Omron CX-Programmer project COREX_92 (CX-Programmer 9.20)
; (V2.0)

# PLC NewPLC1: CJ1G-H CPU42
I/O table (CPU CJ1G-CPU42H): rack 0 slot 0 CJ1W-ID261; rack 0 slot 1 CJ1W-ID261; rack 0 slot 2 CJ1W-OD211; rack 0 slot 3 CJ1W-OD212; rack 0 slot 4 CJ1W-OD212; rack 0 slot 5 CJ1W-OD212; rack 0 slot 6 CJ1W-OD212; rack 0 slot 7 CJ1W-OD212; rack 0 slot 8 CJ1W-AD041-V1

## Global symbols (name address type ; comment)
2000 CHANNEL  ; Peak Value Hold Unitat 0
2001 CHANNEL  ; AIn1 - cèlula aliniador MUW
2002 CHANNEL  ; AIn2 - cèlula ultrassons reb. esquerra
2003 CHANNEL  ; AIn3 - cèlula aliniador reb. dret
2009 CHANNEL  ; Detecció Desconnexió Entrades Unitat 0
2.05 BOOL  ; Relé velocitat màquina mestre
2.06 BOOL  ; màquina mestra unida
2.07 BOOL  ; Info reset de la mestra cap a l'esclava
2.08 BOOL  ; Marxa des de la mestra
2.09 BOOL  ; Mestra en marxa en mode B (Engegada de la mestra)
2.10 BOOL  ; premarxa de la mestra
2.11 BOOL  ; $?St$Bk?_#[971] / mestre en mode "A"$?St$Bk?_#[971]
2.12 BOOL  ; Sèrie de paros de la mestra
2.13 BOOL  ; Màquina mestra en cicle
2.14 BOOL  ; Info SM alt a master
2.15 BOOL  ; Relé velocitat mestra a esclava
30.06 BOOL  ; Sel. Giro Invers MUW
30.07 BOOL  ; Puls.Tensat MUW
320.09 BOOL  ; Tecla calibrar ultrassons MUW
320.10 BOOL  ; Tecla calibrar ultrassons reb.esquerra
320.11 BOOL  ; Tecla calibrar ultrassons reb. dret
32.03 BOOL  ; Alarma variadors de freqüència
32.07 BOOL  ; Marxa aliniador desbobinador
34.13 BOOL  ; Botó negre comanament a distància
36.01 BOOL  ; Selector mode desplaçador (abans selector línia)
36.03 BOOL  ; Detector SM alt master
36.04 BOOL  ; Detector SM de la mestra al mig
36.05 BOOL  ; Detector SM baix master
36.06 BOOL  ; Pulsador marxa lenta SM
36.08 BOOL  ; Detector SM alt esclava
36.09 BOOL  ; Detector SM baix esclava
36.10 BOOL  ; Màquina esclava unida
36.11 BOOL  ; Pulsador de reset de la esclava
36.12 BOOL  ; Condicions premarxa esclava
36.13 BOOL  ; Esclava en premarxa
36.14 BOOL  ; $?St$Bk?_#[972] / esclava en mode "A"$?St$Bk?_#[972]
36.15 BOOL  ; Sèrie de paros de l'esclava
37.00 BOOL  ; Màquina esclava en cicle
4.12 BOOL  ; elv desplaçar a l'esquerra aliniador desbobinador
4.13 BOOL  ; elv desplaçar a la dreta aliniador desbobinador
50.05 BOOL  ; Reset des de l'esclava
50.06 BOOL  ; Impuls reset des de l'esclava
5.06 BOOL  ; Pilot MUW
6.14 BOOL  ; Marxa Inversa MUW
7.08 BOOL  ; elv.desplaçar a l'esquerra aliniador esquerra (destapar)
7.09 BOOL  ; elv.desplaçar a la dreta aliniador esquerra (tapar)
7.10 BOOL  ; elv.desplaçar a l'esquerra aliniador dret (tapar)
7.11 BOOL  ; elv.desplaçar a la dreta aliniador dret (destapar)
7.12 BOOL  ; Marxa normal SM
7.13 BOOL  ; Marxa lenta SM
7.14 BOOL  ; contactor motor bufador SM
80.01 BOOL  ; Estat 1 reb. esquerra
80.02 BOOL  ; Estat2 reb. esquerra
80.03 BOOL  ; Estat3 reb. esquerra
81.01 BOOL  ; Estat 1 reb. dret
81.02 BOOL  ; Estat2 reb. dret
81.03 BOOL  ; Estat3 reb. dret
89.00 BOOL  ; aux. detectors SM alt
89.01 BOOL  ; Aux SM baix
89.02 BOOL  ; Aux SM alt
91.10 BOOL  ; Impuls canvi rotlle rebuig
91.11 BOOL  ; Màquines unides
91.12 BOOL  ; Coincidència selecció entre les dues màquines
91.13 BOOL  ; Missatge cal rearmar la màquina esclava
91.14 BOOL  ; Aux.esclava no està en condicions de marxa
91.15 BOOL  ; Aux.Autogir
92.03 BOOL  ; Aux. MUW OK
9.04 BOOL  ; ZIG-ZAG ESQUERRA
9.05 BOOL  ; ZIG-ZAG DRETA
C0032 BOOL  ; nombre bosses rebuig en engegar
C0150 BOOL  ; pulsos aliniador muw
C0151 BOOL  ; Afegit per a variar el punt esquerra
C0152 BOOL  ; Afegit per a variar el punt dret
C0250 BOOL  ; Bosses fabricades x 1E0
C0251 BOOL  ; Bosses fabricades x 1E4
C0252 BOOL  ; Bosses fabricades x 1E8
C0253 BOOL  ; Rotlles esquerres x 1E0
C0254 BOOL  ; Rotlles esquerres x 1E4
C0255 BOOL  ; Rotlles esquerres x 1E8
C0256 BOOL  ; Rotlles drets x 1E0
C0257 BOOL  ; Rotlles drets x 1E4
C0258 BOOL  ; Rotlles drets x 1E8
C0555 BOOL  ; ret
C151 CHANNEL  ; Afegit per a variar ventall cada cicle
D200 CHANNEL  ; Divisor per a l'entrada ultrassonic MUW
D20000 CHANNEL  ; Habilitar conversions Unitat 0
D20001 CHANNEL  ; Configuracio rangs Unitat 0
D20002 CHANNEL  ; Valor mig entrada 1
D20003 CHANNEL  ; Valor mig entrada 2
D20004 CHANNEL  ; Valor mig entrada 3
D20005 CHANNEL  ; Valor mig entrada 4
D20006 CHANNEL  ; Valor mig entrada 5
D20007 CHANNEL  ; Valor mig entrada 6
D20008 CHANNEL  ; Valor mig entrada 7
D20009 CHANNEL  ; Valor mig entrada 8
D20018 CHANNEL  ; Temps conversió/ressolució unitat0
D201 CHANNEL  ; residu divisió
D202 CHANNEL  ; Divisor per a ultrassonic reb. esquerra
D203 CHANNEL  ; residu divisió
D204 CHANNEL  ; Divisor per a ultrassonic reb. dret
D205 CHANNEL  ; residu divisió
D210 CHANNEL  ; Percentatge de lectura del MUW
D220 CHANNEL  ; Percentatge de lectura del reb. esquerra
D222 CHANNEL  ; Quantitat de ventall esquerra (BCD)
D223 CHANNEL  ; Ventall total a fer reb. esquerra
D230 CHANNEL  ; Percentatge de lectura del reb. dret
D232 CHANNEL  ; Quantitat de ventall dret(BCD)
D233 CHANNEL  ; Ventall total a fer reb. dret
D40 CHANNEL  ; missatge a veure en prova pneumàtica
H0.15 BOOL  ; habilita canvi rotlle de rebuig
T0030 BOOL  ; Fi marxa vibrador esquerra
T0031 BOOL  ; Fi marxa vibrador dreta
T0081 BOOL  ; Retard missatge esclava no preparada
T0150 BOOL  ; retard calibrar ultrasons MUW
T0151 BOOL  ; retard calibrar ultrassons reb.esquerra
T0152 BOOL  ; retard calibrar ultrassons reb. dret
T0153 BOOL  ; retard seguretat moviment brusc aliniador MUW
T0154 BOOL  ; temps mínim elv a esquerres desactivada
T0155 BOOL  ; temps mínim elv a dretes desactivada
T0156 BOOL  ; Temps ventall reb. esquerra
T0157 BOOL  ; Temps Interior esquerra (esperem per destapar)
T0158 BOOL  ; Temps ventall reb. dret
T0159 BOOL  ; Temps Interior dret (esperem per destapar)
T0340 BOOL  ; Temps coincidència entre màquines
T0341 BOOL  ; Bufat allargat SM
T0555 BOOL  ; ret
n120_08 120.08 BOOL  ; MSG.DIGIT.0
n120_09 120.09 BOOL  ; MSG.DIGIT.1
n120_10 120.10 BOOL  ; MSG.DIGIT.2
n120_11 120.11 BOOL  ; MSG.DIGIT.3
n120_12 120.12 BOOL  ; MSG.DIGIT.4
n120_13 120.13 BOOL  ; MSG.DIGIT.5
n120_14 120.14 BOOL  ; MSG.DIGIT.6
n235_05 235.05 BOOL  ; CELUL.ROLL.EN VI
n235_06 235.06 BOOL  ; CELUL.VOLC.VAC.I
n236_05 236.05 BOOL  ; CULUL,ROLL.EN.VD
n236_06 236.06 BOOL  ; CELUL.VOLC.VAC.D
n237_00 237.00 BOOL  ; CELUL.DEP/MDR.I
n237_01 237.01 BOOL  ; CELUL.ASCN.LLN.I
n237_05 237.05 BOOL  ; CELUL.R.CAIDO IZ
n237_08 237.08 BOOL  ; CELUL.DEP/MDR.D
n237_09 237.09 BOOL  ; CELUL.ASCN.LLN.D
n237_13 237.13 BOOL  ; CELUL.R.CAIDO DR
n253_08 A402.04 BOOL  ; LOW BATTERY
n253_13 CF113 BOOL  ; ON.
n253_14 CF114 BOOL  ; OFF.
n253_15 A200.15 BOOL  ; FIRST CYCLE FLAG
n254_00 CF104 BOOL  ; IMP 1Min.
n255_00 CF100 BOOL  ; IMP 0.1Seg.
n255_01 CF101 BOOL  ; IMP 0.2Seg
n255_02 CF102 BOOL  ; IMP 1Seg.
n2_00 2.00 BOOL  ; CONTROL VELO.A.I
n2_01 2.01 BOOL  ; CONTROL VELO.B.I
n2_02 2.02 BOOL  ; CONTROL VELO.A.D
n2_03 2.03 BOOL  ; CONTROL VELO.B.D
n2_04 2.04 BOOL  ; RESET INTEGRADOR
n300_00 300.00 BOOL  ; CAMBIO CICLO
n301_00 301.00 BOOL  ; MARCHA/PARO
n301_01 301.01 BOOL  ; CLOCK
n301_02 301.02 BOOL  ; PULSO FLIP-FLOP
n301_03 301.03 BOOL  ; FLIP-FLOP
n301_04 301.04 BOOL  ; RESET
n301_05 301.05 BOOL  ; SET
n302_00 302.00 BOOL  ; SHFT-PISON
n302_01 302.01 BOOL  ; SHFT-EXTRACTOR
n302_02 302.02 BOOL  ; SHFT-VOLCADOR
n302_03 302.03 BOOL  ; SHFT-ASCENSOR
n302_04 302.04 BOOL  ; SHFT-INTRODUCTOR
n302_05 302.05 BOOL  ; SHFT-SOPLADOR
n302_06 302.06 BOOL  ; SHFT-RESET
n303_11 303.11 BOOL  ; I.CIERRE PISONES
n303_12 303.12 BOOL  ; AUX.C.SOPLADORES
n303_13 303.13 BOOL  ; AUX.C.SOPLADORS
n303_14 303.14 BOOL  ; AUX.A.SOPLADORS
n304_00 304.00 BOOL  ; KEEP PI.NEUMATIC
n305_00 305.00 BOOL  ; KEEP 2PI
n305_01 305.01 BOOL  ; I.REPET.2PI
n307_00 307.00 BOOL  ; I.ABRIR PSN.I.
n307_01 307.01 BOOL  ; I.ABRIR PSN.D.
n307_02 307.02 BOOL  ; I.2PI.ABRIR PSN.
n307_03 307.03 BOOL  ; I.1PI.ABRIR PSN.
n307_04 307.04 BOOL  ; I.1PI.CERRAR PSN
n307_05 307.05 BOOL  ; I.CERR.EXTR.I.
n307_06 307.06 BOOL  ; I.CERR.EXTR.D.
n307_07 307.07 BOOL  ; I.2PI CERR.EXTRC
n307_08 307.08 BOOL  ; I.1PI CERR.EXTRC
n307_09 307.09 BOOL  ; I.ABRIR.EXTRACT
n307_10 307.10 BOOL  ; I.2PI ABRIR EXTR
n307_11 307.11 BOOL  ; I.1PI ABRIR EXTR
n307_12 307.12 BOOL  ; I.ABRIR INTRO.I
n307_13 307.13 BOOL  ; I.ABRIR INTRO.D
n307_14 307.14 BOOL  ; I.2PI ABRIR INTR
n307_15 307.15 BOOL  ; I.1PI ABRIR INTR
n308_00 308.00 BOOL  ; KEEP ABRIR PSN.
n308_01 308.01 BOOL  ; KEEP CERRAR PSN.
n308_02 308.02 BOOL  ; KEEP CERRAR EXTR
n308_03 308.03 BOOL  ; KEEP ABRIR EXTRT
n308_04 308.04 BOOL  ; KEEP ABRIR INTRO
n308_05 308.05 BOOL  ; KEEP ABRIR SOPLD
n308_06 308.06 BOOL  ; KEEP CERRAR SOPD
n308_07 308.07 BOOL  ; KEEP BUFA PEINAR
n308_08 308.08 BOOL  ; KEEP BUFA CORTAR
n308_09 308.09 BOOL  ; KEEP MARCHA PITO
n308_10 308.10 BOOL  ; KEEP PRESOSTATO
n309_00 309.00 BOOL  ; I.ABRIR.SOPLADO
n309_01 309.01 BOOL  ; I.2PI.SOPLADO
n309_02 309.02 BOOL  ; I.1PI.SOPLADO
n309_03 309.03 BOOL  ; I.CERR.SOPLADO
n309_04 309.04 BOOL  ; I.2PI.CERR.SOPLD
n309_05 309.05 BOOL  ; I.1PI.CERR.SOPLD
n309_06 309.06 BOOL  ; I.KEEP B.PEINE
n309_07 309.07 BOOL  ; I.KEEP B.CORTE
n309_08 309.08 BOOL  ; _
n309_09 309.09 BOOL  ; I.ELV.GENERAL
n309_10 309.10 BOOL  ; I.2PI.ELV.GENERL
n309_11 309.11 BOOL  ; I.1PI.ELV.GENERL
n309_12 309.12 BOOL  ; I.PRESOSTATO
n309_13 309.13 BOOL  ; KEEP PITO PRESST
n30_00 30.00 BOOL  ; PARO FIN BOBINA
n30_01 30.01 BOOL  ; AVISO FIN BOBINA
n30_02 30.02 BOOL  ; PARO MAT.CORTADO
n30_03 30.03 BOOL  ; COMP.MUW.ALTO
n30_04 30.04 BOOL  ; COMP.MUW.BAJO
n30_05 30.05 BOOL  ; Sel. Giro Normal MUW
n30_08 30.08 BOOL  ; DETECT.GIRO SR
n30_09 30.09 BOOL  ; MARCHA CALOR SR.
n30_10 30.10 BOOL  ; $?St$Bk?_#[973] / SELECTOR "0" SR.$?St$Bk?_#[973]
n30_11 30.11 BOOL  ; $?St$Bk?_#[974] / SELECTOR "MAN"SR$?St$Bk?_#[974]
n30_12 30.12 BOOL  ; ALARM.TEMPE.SR.
n30_13 30.13 BOOL  ; DETECT.COMP.1
n30_14 30.14 BOOL  ; DETECT.COMP.2
n30_15 30.15 BOOL  ; DETEC.CONTADOR
n310_00 310.00 BOOL  ; PULSO CAMBIO PRG
n310_01 310.01 BOOL  ; KEEP CAMBIO PRG
n311_00 311.00 BOOL  ; I.V.CEL.3505
n311_01 311.01 BOOL  ; I.V.CEL.3506
n311_02 311.02 BOOL  ; I.V.CEL.3605
n311_03 311.03 BOOL  ; I.V.CEL.3606
n311_04 311.04 BOOL  ; I.V.CEL.3700
n311_05 311.05 BOOL  ; I.V.CEL.3701
n311_06 311.06 BOOL  ; I.V.CEL.3705
n311_07 311.07 BOOL  ; I.V.CEL.3708
n311_08 311.08 BOOL  ; I.V.CEL.3709
n311_09 311.09 BOOL  ; I.V.CEL.3713
n311_14 311.14 BOOL  ; KEEP PIT.CEL
n311_15 311.15 BOOL  ; I.PITO.V.CEL
n31_00 31.00 BOOL  ; DET.ALTR.COMP3.I, alrma si no el veu
n31_01 31.01 BOOL  ; DETEC.COMP.I. MEDIO para motors
n31_02 31.02 BOOL  ; PULSAD.GIR.PNZ.I
n31_03 31.03 BOOL  ; DET.ALTR.COMP3.D, alarma si no el veu
n31_04 31.04 BOOL  ; DETEC.COMP.D. MEDIO para motors
n31_05 31.05 BOOL  ; DET.VELO.LINEAL
n31_06 31.06 BOOL  ; PULSAD.GIR.PNZ.D
n31_07 31.07 BOOL  ; PRESOST.CADENAS
n31_08 31.08 BOOL  ; $?St$Bk?_#[975] / SELECT.1-2-4 "1"$?St$Bk?_#[975]
n31_09 31.09 BOOL  ; $?St$Bk?_#[976] / SELECT.1-2-4 "4"$?St$Bk?_#[976]
n31_10 31.10 BOOL  ; SEL.CELUL.REGIST
n31_11 31.11 BOOL  ; PULS.AVANC.REGTR
n31_12 31.12 BOOL  ; PULS.RETRO.REGTR
n31_13 31.13 BOOL  ; SE¥AL REGISTR.OK
n31_14 31.14 BOOL  ; SE¥AL ELV RETROC
n31_15 31.15 BOOL  ; SE¥AL ELV.AVANCE
n320_00 320.00 BOOL  ; TECLA + PRESEL
n320_01 320.01 BOOL  ; TECLA - PRESEL
n320_02 320.02 BOOL  ; TECLA RST PRESEL
n320_03 320.03 BOOL  ; TECLA RST.TOT.R.
n320_04 320.04 BOOL  ; TECLA + PRECAL.
n320_05 320.05 BOOL  ; TECLA - PRECAL.
n320_06 320.06 BOOL  ; TECLA PISTA I
n320_07 320.07 BOOL  ; TECLA PISTA I+D
n320_08 320.08 BOOL  ; TECLA PISTA D
n32_00 32.00 BOOL  ; Emergència Principal OK
n32_01 32.01 BOOL  ; SENYAL RELEs STOPs (Preventa Tapa Tambor)
n32_02 32.02 BOOL  ; Magnetotèrmics i disjuntors
n32_04 32.04 BOOL  ; PRESOSTATO
n32_05 32.05 BOOL  ; AJUST.NIV.COMP3I
n32_06 32.06 BOOL  ; AJUST.NIV.COMP3D
n32_08 32.08 BOOL  ; $?St$Bk?_#[977] / SELECT.MODO"A-B"$?St$Bk?_#[977]
n32_09 32.09 BOOL  ; PULSD.RESTART
n32_10 32.10 BOOL  ; PULSD.RESET
n32_11 32.11 BOOL  ; PULSAD.MARCHA
n32_12 32.12 BOOL  ; PULSAD.PARO
n32_13 32.13 BOOL  ; PULSAD.GIR.TAMB.
n32_14 32.14 BOOL  ; ALARMA RESISTRON
n33_00 33.00 BOOL  ; DETEC.C.PISN.I.C
n33_01 33.01 BOOL  ; DETEC.MAX.ROLL.I
n33_02 33.02 BOOL  ; DETEC.C.EXTR.I.A
n33_03 33.03 BOOL  ; DETEC.C.EXTR.I.C
n33_04 33.04 BOOL  ; CELUL.ROLL.EN VI
n33_05 33.05 BOOL  ; CELUL.VOLC.VAC.I
n33_06 33.06 BOOL  ; DETEC.EJE/MNDR.I
n33_07 33.07 BOOL  ; CELUL.DEP/MDR.I
n33_08 33.08 BOOL  ; CELUL.ASCN.LLN.I
n33_09 33.09 BOOL  ; DETEC.C.INTR.I.A
n33_10 33.10 BOOL  ; CELUL.R.CAIDO IZ
n33_11 33.11 BOOL  ; DETEC.C.PISN.D.C
n33_12 33.12 BOOL  ; DETEC.MAX.ROLL.D
n33_13 33.13 BOOL  ; DETEC.C.EXTR.D.A
n33_14 33.14 BOOL  ; DETEC.C.EXTR.D.C
n33_15 33.15 BOOL  ; CULUL,ROLL.EN.VD
n34_00 34.00 BOOL  ; CELUL.VOLC.VAC.D
n34_01 34.01 BOOL  ; DETEC.EJE/MNDR.D
n34_02 34.02 BOOL  ; DETEC.C.SOPLAD.A
n34_03 34.03 BOOL  ; DETEC.C.SOPLAD.C
n34_04 34.04 BOOL  ; CELUL.DEP/MDR.D
n34_05 34.05 BOOL  ; CELUL.ASCN.LLN.D
n34_06 34.06 BOOL  ; DETEC.C.INTR.D.A
n34_07 34.07 BOOL  ; CELUL.R.CAIDO DR
n34_08 34.08 BOOL  ; DETEC.PARO TAMB.
n34_09 34.09 BOOL  ; DETEC.CUADR.TAMB
n34_10 34.10 BOOL  ; DETEC.POSIC.TAMB
n35_00 35.00 BOOL  ; SELEC.MARCHA F.B
n35_01 35.01 BOOL  ; DETECT.F.B.ALTO
n35_02 35.02 BOOL  ; DETECT.F.B.BAJO
n35_03 35.03 BOOL  ; P.MARCH.LENTA FB
n3_00 3.00 BOOL  ; ELV.S.R.
n3_01 3.01 BOOL  ; ELV.SOPLAD.TAMBR
n3_02 3.02 BOOL  ; ELV.ASCENSOR A.I
n3_03 3.03 BOOL  ; ELV.ASCENSOR C.I
n3_04 3.04 BOOL  ; ELV.INTRODUC.A.I
n3_05 3.05 BOOL  ; ELV.INTRODUC.C.I
n3_06 3.06 BOOL  ; ELV. PISON A.I.
n3_07 3.07 BOOL  ; ELV.PISON C.I.
n3_08 3.08 BOOL  ; ELV.EXTRACT.A.I.
n3_09 3.09 BOOL  ; ELV.EXTRACT.C.I.
n3_10 3.10 BOOL  ; ELV.VOLCD.A.I.
n3_11 3.11 BOOL  ; ELV.VOLCD.C.I.
n3_12 3.12 BOOL  ; ELV.SOPLADOR I.
n3_13 3.13 BOOL  ; ELV.BAR SOPLAD.A
n3_14 3.14 BOOL  ; ELV.BAR.SOPLAD.C
n3_15 3.15 BOOL  ; ELV.ACERCADORES
n41_00 41.00 BOOL  ; PRE.POSC-GIR.TAM
n41_01 41.01 BOOL  ; AUX.G.MAN.TAMBOR
n41_02 41.02 BOOL  ; I.POSIC.CILINDRS
n41_03 41.03 BOOL  ; GIRO AUTO TAMBOR
n41_04 41.04 BOOL  ; DETEC.POSICIONAD
n41_05 41.05 BOOL  ; PRE-POSICIONADO
n41_06 41.06 BOOL  ; CLAXON GIRO.TAMB
n41_07 41.07 BOOL  ; PRE-POS.CILINDRO
n41_08 41.08 BOOL  ; CLAXON PREPOS.CL
n42_00 42.00 BOOL  ; CONDIC. EN 0
n42_01 42.01 BOOL  ; CONDIC.EN 2
n42_02 42.02 BOOL  ; I.POSICION TAMB.
n42_03 42.03 BOOL  ; I.EXTRC.PREMARCH
n42_04 42.04 BOOL  ; I.FI.G/TAMBOR
n42_05 42.05 BOOL  ; I.PIS+SOPL.CERRD
n42_06 42.06 BOOL  ; CONDIC.EN 9
n42_07 42.07 BOOL  ; CONDIC.EN 10
n42_08 42.08 BOOL  ; MF.CAX.GIR.TAMB
n42_09 42.09 BOOL  ; MF.CAX.VIBRD.IZD
n42_10 42.10 BOOL  ; MF.CAX.VIBRAD.DR
n42_11 42.11 BOOL  ; CLAX.DEPOSITOS V
n42_15 42.15 BOOL  ; AUX PULD.GIR.TAM
n43_00 43.00 BOOL  ; I.DETEC.C.EXTR.I
n43_01 43.01 BOOL  ; AUX.RET.EXT.I.
n43_02 43.02 BOOL  ; I.RET.EXTRAC.I.
n43_03 43.03 BOOL  ; I.DET.C.EXTRC.D.
n43_04 43.04 BOOL  ; AUX.RET.EXTRAC.D
n43_05 43.05 BOOL  ; I.RET.EXTRAC.D.
n43_06 43.06 BOOL  ; MEMO.MANDRIL IZ.
n43_07 43.07 BOOL  ; I.INTROD.MANDR.I
n43_08 43.08 BOOL  ; MEMO.MANDRIL D.
n43_09 43.09 BOOL  ; I.INTRD.MANDR.D.
n43_10 43.10 BOOL  ; I.IN.MANDRIL IZD
n43_11 43.11 BOOL  ; AUX.RETRO.MAND.I
n43_12 43.12 BOOL  ; I.INTR.MANDR.I
n43_13 43.13 BOOL  ; I.MANDR.DRH.
n43_14 43.14 BOOL  ; AUX.IN.MAND.DR.
n43_15 43.15 BOOL  ; I.RETR.MANDR.DR.
n44_00 44.00 BOOL  ; AUX.ASCENSOR IZ.
n44_01 44.01 BOOL  ; I.SUB.ASC.IZ
n44_02 44.02 BOOL  ; I.BAJ.ASC.IZ.
n44_03 44.03 BOOL  ; AVIS.FALT.MNDR.I
n44_05 44.05 BOOL  ; AUX.ASCENSOR DRH
n44_06 44.06 BOOL  ; I.SUB.ASC.DRCH.
n44_07 44.07 BOOL  ; I.BAJ.ASC.DRCH
n44_08 44.08 BOOL  ; AVIS.FALT.MNDR.D
n44_12 44.12 BOOL  ; TOPE ASCEN.IZD.
n44_13 44.13 BOOL  ; TOPE ASCEN.DRCH.
n45_00 45.00 BOOL  ; $?St$Bk?_#[978] / INDICA CICLO "A"$?St$Bk?_#[978]
n45_01 45.01 BOOL  ; HASTA A2 I
n45_02 45.02 BOOL  ; HASTA A2 D.
n45_03 45.03 BOOL  ; HASTA A3
n45_04 45.04 BOOL  ; HASTA A4 I
n45_05 45.05 BOOL  ; HASTA A4 D
n45_06 45.06 BOOL  ; HASTA A5
n45_07 45.07 BOOL  ; $?St$Bk?_#[979] / GIRO EN "A"$?St$Bk?_#[979]
n45_08 45.08 BOOL  ; I.FIN GIRO TAMB.
n46_01 46.01 BOOL  ; EN A2 I
n46_02 46.02 BOOL  ; EN A2 D
n46_03 46.03 BOOL  ; EN A4 I
n46_04 46.04 BOOL  ; EN A4 D
n47_00 47.00 BOOL  ; I.ABR.PIS Y SOPL
n47_01 47.01 BOOL  ; I.VOLCA IZD.
n47_02 47.02 BOOL  ; I.VOLCA.DRC.
n47_03 47.03 BOOL  ; I.EXTRACTOR
n47_04 47.04 BOOL  ; I.INTRO.IZD.
n47_05 47.05 BOOL  ; I.INTRO.DRCH
n47_06 47.06 BOOL  ; $?St$Bk?_#[980] / I.FIN CICLO "A"$?St$Bk?_#[980]
n48_00 48.00 BOOL  ; INDICA CICLO B
n48_01 48.01 BOOL  ; I.ABR.PIS Y SOPL
n48_03 48.03 BOOL  ; HASTA B2
n48_04 48.04 BOOL  ; GIRO EN B
n48_10 48.10 BOOL  ; IMPULSO CARGA
n48_11 48.11 BOOL  ; CLOCK
n48_12 48.12 BOOL  ; KEEP IMPULSO RES
n48_13 48.13 BOOL  ; IMP.RESET CONTAD
n49_00 49.00 BOOL  ; I.ABR.VOLCD.IZ
n49_01 49.01 BOOL  ; I.CERR.VOLCD.IZD
n49_02 49.02 BOOL  ; I.ABR.VOLCD.DRH
n49_03 49.03 BOOL  ; I.CERR.VOLCD.DRC
n4_00 4.00 BOOL  ; ELV.ASCEMSOR A.D
n4_01 4.01 BOOL  ; ELV.ASCENSOR C.D
n4_02 4.02 BOOL  ; ELV.INTRODUC.A.D
n4_03 4.03 BOOL  ; ELV.INTRODUC.C.D
n4_04 4.04 BOOL  ; ELV.PISON A.D.
n4_05 4.05 BOOL  ; ELV.PISON C.D.
n4_06 4.06 BOOL  ; ELV.EXTRACT.A.D.
n4_07 4.07 BOOL  ; ELV.EXTRACT.C.D.
n4_08 4.08 BOOL  ; ELV.PRE-SOPLADO
n4_09 4.09 BOOL  ; ELV.VOLCD.A.D.
n4_10 4.10 BOOL  ; ELV.VOLCD.C.D.
n4_11 4.11 BOOL  ; ELV.SOPLADOR D.
n4_14 4.14 BOOL  ; ELV.AVANC.IMPRES
n4_15 4.15 BOOL  ; ELV.RETRO.IMPRES
n50_00 50.00 BOOL  ; IMPULSO RESET
n50_01 50.01 BOOL  ; TEST.PILOTOS
n50_10 50.10 BOOL  ; AUX.NO REGISTRO
n50_11 50.11 BOOL  ; AUX.PLT.CEL.REGS
n50_12 50.12 BOOL  ; AUX.PLT.REGIS.OK
n50_13 50.13 BOOL  ; AUX.ENCLAV.REGST
n51_00 51.00 BOOL  ; AUX.PILOTO L.B.
n51_01 51.01 BOOL  ; PULSOS LOW BATT.
n51_02 51.02 BOOL  ; AUX.CLAXON LOW.B
n51_04 51.04 BOOL  ; AUX.PLT.MAQUINA
n51_06 51.06 BOOL  ; AUX.PLT.C/ROLLO
n52_01 52.01 BOOL  ; SUMA MF.CAX.
n53_00 53.00 BOOL  ; K.HABILIT.A.IZD
n53_01 53.01 BOOL  ; K.FRENO A IZD.
n53_02 53.02 BOOL  ; K.HABILIT.B.IZD.
n53_03 53.03 BOOL  ; K.FRENO B.IZD.
n53_04 53.04 BOOL  ; K.HABILIT.A.DRH.
n53_05 53.05 BOOL  ; K.FRENO A.DRCH
n53_06 53.06 BOOL  ; K.HABILIT.B.DRCH
n53_07 53.07 BOOL  ; K.FRENO B.DRCH
n53_08 53.08 BOOL  ; V.TANGEN.A.I+D
n53_09 53.09 BOOL  ; V.TANGEN.B.I+D
n53_10 53.10 BOOL  ; CND.JOG.MOT.REBO
n53_11 53.11 BOOL  ; AUX.JOG.A.IZD
n53_12 53.12 BOOL  ; AUX.JOG.B.IZD.
n53_13 53.13 BOOL  ; AUX.JOG.A.DRCH.
n53_14 53.14 BOOL  ; AUX.JOG.B.DRCH.
n53_15 53.15 BOOL  ; AUX.RET.PARO REB
n5_00 5.00 BOOL  ; PILOTO MANIOBRA
n5_01 5.01 BOOL  ; PILOTO STOP
n5_02 5.02 BOOL  ; PILOTO MAQ.OK.
n5_03 5.03 BOOL  ; PILOTO C/ROLLO
n5_04 5.04 BOOL  ; PLT.ROLL.NO CAID
n5_05 5.05 BOOL  ; CLAXON
n5_07 5.07 BOOL  ; XENO FLASH
n5_08 5.08 BOOL  ; PLT.REGISTRO OK
n5_09 5.09 BOOL  ; MARCHA NORM F.B.
n5_10 5.10 BOOL  ; MARCHA LENT.F.B.
n60_00 60.00 BOOL  ; MSG  0
n60_01 60.01 BOOL  ; MSG  1
n60_02 60.02 BOOL  ; MSG  2
n60_03 60.03 BOOL  ; MSG  3
n60_04 60.04 BOOL  ; MSG  4
n60_05 60.05 BOOL  ; MSG  5
n60_06 60.06 BOOL  ; MSG  6
n60_07 60.07 BOOL  ; MSG  7
n60_08 60.08 BOOL  ; MSG  8
n60_09 60.09 BOOL  ; MSG  9
n60_10 60.10 BOOL  ; MSG 10
n60_11 60.11 BOOL  ; MSG 11
n60_12 60.12 BOOL  ; MSG 12
n60_13 60.13 BOOL  ; MSG 13
n60_14 60.14 BOOL  ; MSG 14
n60_15 60.15 BOOL  ; MSG 15
n61_00 61.00 BOOL  ; MSG 16
n61_01 61.01 BOOL  ; MSG 17
n61_02 61.02 BOOL  ; MSG 18
n61_03 61.03 BOOL  ; MSG 19
n61_04 61.04 BOOL  ; MSG 20
n61_05 61.05 BOOL  ; MSG 21
n61_06 61.06 BOOL  ; MSG 22
n61_07 61.07 BOOL  ; MSG 23
n61_08 61.08 BOOL  ; MSG 24
n61_09 61.09 BOOL  ; MSG 25
n61_10 61.10 BOOL  ; MSG 26
n61_11 61.11 BOOL  ; MSG 27
n61_12 61.12 BOOL  ; MSG 28
n61_13 61.13 BOOL  ; MSG 29
n61_14 61.14 BOOL  ; MSG 30
n61_15 61.15 BOOL  ; MSG 31
n62_00 62.00 BOOL  ; MSG 32
n62_01 62.01 BOOL  ; MSG 33
n62_02 62.02 BOOL  ; MSG 34
n62_03 62.03 BOOL  ; MSG 35
n62_04 62.04 BOOL  ; MSG 36
n62_05 62.05 BOOL  ; MSG 37
n62_06 62.06 BOOL  ; MSG 38
n62_07 62.07 BOOL  ; MSG 39
n62_08 62.08 BOOL  ; MSG 40
n62_09 62.09 BOOL  ; MSG 41
n62_10 62.10 BOOL  ; MSG 42
n62_11 62.11 BOOL  ; MSG 43
n62_12 62.12 BOOL  ; MSG 44
n62_13 62.13 BOOL  ; MSG 45
n62_14 62.14 BOOL  ; MSG 46
n62_15 62.15 BOOL  ; MSG 47
n63_00 63.00 BOOL  ; MSG 48
n63_01 63.01 BOOL  ; MSG 49
n63_02 63.02 BOOL  ; MSG 50
n63_03 63.03 BOOL  ; MSG 51
n63_04 63.04 BOOL  ; MSG 52
n63_05 63.05 BOOL  ; MSG 53
n63_06 63.06 BOOL  ; MSG 54
n63_07 63.07 BOOL  ; MSG 55
n63_08 63.08 BOOL  ; MSG 56
n63_09 63.09 BOOL  ; MSG 57
n63_10 63.10 BOOL  ; MSG 58
n63_11 63.11 BOOL  ; MSG 59
n63_12 63.12 BOOL  ; MSG 60
n63_13 63.13 BOOL  ; MSG 61
n63_14 63.14 BOOL  ; MSG 62
n63_15 63.15 BOOL  ; MSG 63
n64_00 64.00 BOOL  ; MSG 64
n64_01 64.01 BOOL  ; MSG 65
n64_02 64.02 BOOL  ; MSG 66
n64_03 64.03 BOOL  ; MSG 67
n64_04 64.04 BOOL  ; MSG 68
n64_05 64.05 BOOL  ; MSG 69
n64_06 64.06 BOOL  ; MSG 70
n64_07 64.07 BOOL  ; MSG 71
n64_08 64.08 BOOL  ; MSG 72
n64_09 64.09 BOOL  ; MSG 73
n64_10 64.10 BOOL  ; MSG 74
n64_11 64.11 BOOL  ; MSG 75
n64_12 64.12 BOOL  ; MSG 76
n64_13 64.13 BOOL  ; MSG 77
n64_14 64.14 BOOL  ; MSG 78
n64_15 64.15 BOOL  ; MSG 79
n65_00 65.00 BOOL  ; MSG 80
n65_01 65.01 BOOL  ; MSG 81
n65_02 65.02 BOOL  ; MSG 82
n65_03 65.03 BOOL  ; MSG 83
n65_04 65.04 BOOL  ; MSG 84
n65_05 65.05 BOOL  ; MSG 85
n65_06 65.06 BOOL  ; MSG 86
n65_07 65.07 BOOL  ; MSG 87
n65_08 65.08 BOOL  ; MSG 88
n65_09 65.09 BOOL  ; MSG 89
n65_10 65.10 BOOL  ; MSG 90
n65_11 65.11 BOOL  ; MSG 91
n65_12 65.12 BOOL  ; MSG 92
n65_13 65.13 BOOL  ; MSG 93
n65_14 65.14 BOOL  ; MSG 94
n65_15 65.15 BOOL  ; MSG 95
n66_00 66.00 BOOL  ; MSG 96
n66_01 66.01 BOOL  ; MSG 97
n66_02 66.02 BOOL  ; MSG 98
n66_03 66.03 BOOL  ; MSG 99
n66_04 66.04 BOOL  ; MSG 100
n66_05 66.05 BOOL  ; MSG 101
n66_06 66.06 BOOL  ; MSG 102
n66_07 66.07 BOOL  ; MSG 103
n66_08 66.08 BOOL  ; MSG 104
n66_09 66.09 BOOL  ; MSG 105
n66_10 66.10 BOOL  ; MSG 106
n66_11 66.11 BOOL  ; MSG 107
n66_12 66.12 BOOL  ; MSG 108
n66_13 66.13 BOOL  ; MSG 109
n66_14 66.14 BOOL  ; MSG 110
n66_15 66.15 BOOL  ; MSG 111
n67_00 67.00 BOOL  ; MSG 112
n67_01 67.01 BOOL  ; MSG 113
n67_02 67.02 BOOL  ; MSG 114
n67_03 67.03 BOOL  ; MSG 115
n67_04 67.04 BOOL  ; MSG 116
n67_05 67.05 BOOL  ; MSG 117
n67_06 67.06 BOOL  ; MSG 118
n67_07 67.07 BOOL  ; MSG 119
n67_08 67.08 BOOL  ; MSG 120
n67_09 67.09 BOOL  ; MSG 121
n67_10 67.10 BOOL  ; MSG 122
n67_11 67.11 BOOL  ; MSG 123
n67_12 67.12 BOOL  ; MSG 124
n67_13 67.13 BOOL  ; MSG 125
n67_14 67.14 BOOL  ; MSG 126
n67_15 67.15 BOOL  ; MSG 127
n68_00 68.00 BOOL  ; MSG 128
n68_01 68.01 BOOL  ; RESERVADO MSGS.
n68_02 68.02 BOOL  ; RESERVADO MSGS.
n68_03 68.03 BOOL  ; RESERVADO MSGS.
n68_04 68.04 BOOL  ; RESERVADO MSGS.
n68_05 68.05 BOOL  ; RESERVADO MSGS.
n68_06 68.06 BOOL  ; RESERVADO MSGS.
n68_07 68.07 BOOL  ; RESERVADO MSGS.
n68_08 68.08 BOOL  ; RESERVADO MSGS.
n68_09 68.09 BOOL  ; RESERVADO MSGS.
n68_10 68.10 BOOL  ; RESERVADO MSGS.
n68_11 68.11 BOOL  ; RESERVADO MSGS.
n68_12 68.12 BOOL  ; RESERVADO MSGS.
n68_13 68.13 BOOL  ; RESERVADO MSGS.
n68_14 68.14 BOOL  ; RESERVADO MSGS.
n68_15 68.15 BOOL  ; RESERVADO MSGS.
n69_00 69.00 BOOL  ; RESERVADO MSGS.
n69_01 69.01 BOOL  ; RESERVADO MSGS.
n69_02 69.02 BOOL  ; RESERVADO MSGS.
n69_03 69.03 BOOL  ; RESERVADO MSGS.
n69_04 69.04 BOOL  ; RESERVADO MSGS.
n69_05 69.05 BOOL  ; RESERVADO MSGS.
n69_06 69.06 BOOL  ; RESERVADO MSGS.
n69_07 69.07 BOOL  ; RESERVADO MSGS.
n69_08 69.08 BOOL  ; RESERVADO MSGS.
n69_09 69.09 BOOL  ; RESERVADO MSGS.
n69_10 69.10 BOOL  ; RESERVADO MSGS.
n69_11 69.11 BOOL  ; RESERVADO MSGS.
n69_12 69.12 BOOL  ; RESERVADO MSGS.
n69_13 69.13 BOOL  ; RESERVADO MSGS.
n69_14 69.14 BOOL  ; RESERVADO MSGS.
n69_15 69.15 BOOL  ; RESERVADO MSGS.
n6_00 6.00 BOOL  ; CONTROL DIG.1A.I
n6_01 6.01 BOOL  ; CONTROL DIG.2A.I
n6_02 6.02 BOOL  ; CONTROL DIG.3A.I
n6_03 6.03 BOOL  ; CONTROL DIG.1B.I
n6_04 6.04 BOOL  ; CONTROL DIG.2B.I
n6_05 6.05 BOOL  ; CONTROL DIG.3B.I
n6_06 6.06 BOOL  ; CONTROL DIG.1A.D
n6_07 6.07 BOOL  ; CONTROL DIG.2A.D
n6_08 6.08 BOOL  ; CONTROL DIG.3A.D
n6_09 6.09 BOOL  ; CONTROL DIG.1B.D
n6_10 6.10 BOOL  ; CONTROL DIG.2B.D
n6_11 6.11 BOOL  ; CONTROL DIG.3B.D
n6_12 6.12 BOOL  ; MARCHA LENTA MUW
n6_13 6.13 BOOL  ; MARCHA NORMAL MW
n6_15 6.15 BOOL  ; MARCHA RESISTRON
n70_00 70.00 BOOL  ; RESERVADO MSGS.
n70_01 70.01 BOOL  ; RESERVADO MSGS.
n70_02 70.02 BOOL  ; RESERVADO MSGS.
n70_03 70.03 BOOL  ; RESERVADO MSGS.
n70_04 70.04 BOOL  ; RESERVADO MSGS.
n70_05 70.05 BOOL  ; RESERVADO MSGS.
n70_06 70.06 BOOL  ; RESERVADO MSGS.
n70_07 70.07 BOOL  ; RESERVADO MSGS.
n70_08 70.08 BOOL  ; RESERVADO MSGS.
n70_09 70.09 BOOL  ; RESERVADO MSGS.
n70_10 70.10 BOOL  ; RESERVADO MSGS.
n70_11 70.11 BOOL  ; RESERVADO MSGS.
n70_12 70.12 BOOL  ; RESERVADO MSGS.
n70_13 70.13 BOOL  ; RESERVADO MSGS.
n70_14 70.14 BOOL  ; RESERVADO MSGS.
n70_15 70.15 BOOL  ; RESERVADO MSGS.
n71_00 71.00 BOOL  ; RESERVADO MSGS.
n71_01 71.01 BOOL  ; RESERVADO MSGS.
n71_02 71.02 BOOL  ; RESERVADO MSGS.
n71_03 71.03 BOOL  ; RESERVADO MSGS.
n71_04 71.04 BOOL  ; RESERVADO MSGS.
n71_05 71.05 BOOL  ; RESERVADO MSGS.
n71_06 71.06 BOOL  ; RESERVADO MSGS.
n71_07 71.07 BOOL  ; RESERVADO MSGS.
n71_08 71.08 BOOL  ; RESERVADO MSGS.
n71_09 71.09 BOOL  ; RESERVADO MSGS.
n71_10 71.10 BOOL  ; RESERVADO MSGS.
n71_11 71.11 BOOL  ; RESERVADO MSGS.
n71_12 71.12 BOOL  ; RESERVADO MSGS.
n71_13 71.13 BOOL  ; RESERVADO MSGS.
n71_14 71.14 BOOL  ; RESERVADO MSGS.
n71_15 71.15 BOOL  ; RESERVADO MSGS.
n72_00 72.00 BOOL  ; RESERVADO MSGS.
n72_01 72.01 BOOL  ; RESERVADO MSGS.
n72_02 72.02 BOOL  ; RESERVADO MSGS.
n72_03 72.03 BOOL  ; RESERVADO MSGS.
n72_04 72.04 BOOL  ; RESERVADO MSGS.
n72_05 72.05 BOOL  ; RESERVADO MSGS.
n72_06 72.06 BOOL  ; RESERVADO MSGS.
n72_07 72.07 BOOL  ; RESERVADO MSGS.
n72_08 72.08 BOOL  ; RESERVADO MSGS.
n72_09 72.09 BOOL  ; RESERVADO MSGS.
n72_10 72.10 BOOL  ; RESERVADO MSGS.
n72_11 72.11 BOOL  ; RESERVADO MSGS.
n72_12 72.12 BOOL  ; RESERVADO MSGS.
n72_13 72.13 BOOL  ; RESERVADO MSGS.
n72_14 72.14 BOOL  ; RESERVADO MSGS.
n72_15 72.15 BOOL  ; RESERVADO MSGS.
n73_00 73.00 BOOL  ; RESERVADO MSGS.
n73_01 73.01 BOOL  ; RESERVADO MSGS.
n73_02 73.02 BOOL  ; RESERVADO MSGS.
n73_03 73.03 BOOL  ; RESERVADO MSGS.
n73_04 73.04 BOOL  ; RESERVADO MSGS.
n73_05 73.05 BOOL  ; RESERVADO MSGS.
n73_06 73.06 BOOL  ; RESERVADO MSGS.
n73_07 73.07 BOOL  ; RESERVADO MSGS.
n73_08 73.08 BOOL  ; RESERVADO MSGS.
n73_09 73.09 BOOL  ; RESERVADO MSGS.
n73_10 73.10 BOOL  ; RESERVADO MSGS.
n73_11 73.11 BOOL  ; RESERVADO MSGS.
n73_12 73.12 BOOL  ; RESERVADO MSGS.
n73_13 73.13 BOOL  ; RESERVADO MSGS.
n73_14 73.14 BOOL  ; RESERVADO MSGS.
n73_15 73.15 BOOL  ; RESERVADO MSGS.
n74_00 74.00 BOOL  ; RESERVADO MSGS.
n74_01 74.01 BOOL  ; RESERVADO MSGS.
n74_02 74.02 BOOL  ; RESERVADO MSGS.
n74_03 74.03 BOOL  ; RESERVADO MSGS.
n74_04 74.04 BOOL  ; RESERVADO MSGS.
n74_05 74.05 BOOL  ; RESERVADO MSGS.
n74_06 74.06 BOOL  ; RESERVADO MSGS.
n74_07 74.07 BOOL  ; RESERVADO MSGS.
n74_08 74.08 BOOL  ; RESERVADO MSGS.
n74_09 74.09 BOOL  ; RESERVADO MSGS.
n74_10 74.10 BOOL  ; RESERVADO MSGS.
n74_11 74.11 BOOL  ; RESERVADO MSGS.
n74_12 74.12 BOOL  ; RESERVADO MSGS.
n74_13 74.13 BOOL  ; RESERVADO MSGS.
n74_14 74.14 BOOL  ; RESERVADO MSGS.
n74_15 74.15 BOOL  ; RESERVADO MSGS.
n75_00 75.00 BOOL  ; RESERVADO MSGS.
n75_01 75.01 BOOL  ; RESERVADO MSGS.
n75_02 75.02 BOOL  ; RESERVADO MSGS.
n75_03 75.03 BOOL  ; RESERVADO MSGS.
n75_04 75.04 BOOL  ; RESERVADO MSGS.
n75_05 75.05 BOOL  ; RESERVADO MSGS.
n75_06 75.06 BOOL  ; RESERVADO MSGS.
n75_07 75.07 BOOL  ; RESERVADO MSGS.
n75_08 75.08 BOOL  ; RESERVADO MSGS.
n75_09 75.09 BOOL  ; RESERVADO MSGS.
n75_10 75.10 BOOL  ; RESERVADO MSGS.
n75_11 75.11 BOOL  ; RESERVADO MSGS.
n75_12 75.12 BOOL  ; RESERVADO MSGS.
n75_13 75.13 BOOL  ; RESERVADO MSGS.
n75_14 75.14 BOOL  ; RESERVADO MSGS.
n75_15 75.15 BOOL  ; RESERVADO MSGS.
n76_00 76.00 BOOL  ; AUX.MPX.MSGS.
n76_01 76.01 BOOL  ; AUX.MPX.MSGS.
n76_02 76.02 BOOL  ; AUX.MPX.MSGS.
n76_03 76.03 BOOL  ; AUX.MPX.MSGS.
n76_04 76.04 BOOL  ; AUX.MPX.MSGS.
n76_05 76.05 BOOL  ; AUX.MPX.MSGS.
n76_06 76.06 BOOL  ; AUX.MPX.MSGS.
n76_07 76.07 BOOL  ; AUX.MPX.MSGS.
n76_08 76.08 BOOL  ; AUX.MPX.MSGS.
n76_09 76.09 BOOL  ; AUX.MPX.MSGS.
n76_10 76.10 BOOL  ; AUX.MPX.MSGS.
n76_11 76.11 BOOL  ; AUX.MPX.MSGS.
n76_12 76.12 BOOL  ; AUX.MPX.MSGS.
n76_13 76.13 BOOL  ; AUX.MPX.MSGS.
n76_14 76.14 BOOL  ; AUX.MPX.MSGS.
n76_15 76.15 BOOL  ; AUX.MPX.MSGS.
n7_00 7.00 BOOL  ; MARCHA MAQUINA
n7_01 7.01 BOOL  ; JOG.MAQUINA
n7_02 7.02 BOOL  ; Velocitat per a 2 soldadors
n7_03 7.03 BOOL  ; COTRL.TACO.x1
n7_04 7.04 BOOL  ; COTRL.TACO.x2
n7_05 7.05 BOOL  ; CNT.GIRO TAMBOR
n7_06 7.06 BOOL  ; CNT.VIBRAD.IZD.
n7_07 7.07 BOOL  ; CNT.VIBRAD.DRCH.
n89_03 89.03 BOOL  ; STOP GENERAL
n89_04 89.04 BOOL  ; AUX.PLT.STOPS
n89_05 89.05 BOOL  ; AUX.MSG.AIRE MAN
n89_06 89.06 BOOL  ; MSG.RET.SUB.AIRE
n89_08 89.08 BOOL  ; AUX.AIRE OK
n89_09 89.09 BOOL  ; Missatge Pressió d'aire
n89_12 89.12 BOOL  ; AUX.ESPERE PLS
n89_15 89.15 BOOL  ; KEEP AIRE INI.OK (Pujada d'aire OK)
n90_00 90.00 BOOL  ; AUX.STOP PULSADO
n90_01 90.01 BOOL  ; Magnetotèrmics
n90_02 90.02 BOOL  ; Inverters OK
n90_04 90.04 BOOL  ; SELEC 1 SOLD.
n90_05 90.05 BOOL  ; SELEC.2 SOLD.
n90_06 90.06 BOOL  ; SELEC.4 SOLD.
n90_07 90.07 BOOL  ; AUX.COMP.1
n90_08 90.08 BOOL  ; AUX.COMP.2
n90_09 90.09 BOOL  ; AUX.COMP.3 I.
n90_10 90.10 BOOL  ; AUX.COMP.3 D.
n90_11 90.11 BOOL  ; AUX.TRANS.TAMBOR
n90_14 90.14 BOOL  ; IMP.FIN.TOT.CICL
n90_15 90.15 BOOL  ; MONITOR CICLO
n91_00 91.00 BOOL  ; NIVEL 0
n91_01 91.01 BOOL  ; NIVEL 1
n91_02 91.02 BOOL  ; NIVEL 2
n91_03 91.03 BOOL  ; NIVEL 3
n91_04 91.04 BOOL  ; NIVEL 4
n91_05 91.05 BOOL  ; NIVEL 5
n91_06 91.06 BOOL  ; NIVEL 6
n92_00 92.00 BOOL  ; AUX.FIN BOBINA
n92_01 92.01 BOOL  ; AUX.CLAX.FI.BOB.
n92_02 92.02 BOOL  ; AUX.F.B.ALTO
n92_04 92.04 BOOL  ; AUX.MUW ALTO
n92_05 92.05 BOOL  ; IMP.IN.DETEC.GIR
n92_06 92.06 BOOL  ; IMP.OU.DETEC.GIR
n92_09 92.09 BOOL  ; IND.MOV.MATERIAL
n92_10 92.10 BOOL  ; AUX.POSIC.C3.IU
n92_11 92.11 BOOL  ; AUX.POSIC.C3.ID
n92_12 92.12 BOOL  ; AUX.POSIC.C3.DU
n92_13 92.13 BOOL  ; AUX.POSIC.C3.DD
n92_14 92.14 BOOL  ; K.AVIS.POSIC.C3
n92_15 92.15 BOOL  ; AUX.CLAXON C3
n93_00 93.00 BOOL  ; AUX ALRMTEMP.SR.
n93_01 93.01 BOOL  ; I.DETC.EXTR.AB.I
n93_02 93.02 BOOL  ; AUX.RESET.CAID.I
n93_03 93.03 BOOL  ; MEMO.ROLL.CAID.I
n93_04 93.04 BOOL  ; AUX.MSG.CAIDO.IZ
n93_05 93.05 BOOL  ; I.DETC.EXTR.AB.D
n93_06 93.06 BOOL  ; AUX.RESET CAID.D
n93_07 93.07 BOOL  ; MEMO.ROLL.CAID.D
n93_08 93.08 BOOL  ; AUX.MSG.CAIDO.DR
n93_09 93.09 BOOL  ; CLXON.CAIDA ROLL
n93_10 93.10 BOOL  ; I.IDA EXTRACC.I
n93_11 93.11 BOOL  ; SEGURO EXTRACC.I
n93_12 93.12 BOOL  ; I.IDA EXTRACC.D
n93_13 93.13 BOOL  ; SEGURO EXTRACC.D
n93_14 93.14 BOOL  ; AUX.PLT.ROLL.N/C
n93_15 93.15 BOOL  ; I.CAMBIO IDIOMA
n94_03 94.03 BOOL  ; PISTA IZD.ACTIVA
n94_04 94.04 BOOL  ; PISTA DRH.ACTIVA
n95_00 95.00 BOOL  ; K.PARO EN POSIC.
n95_04 95.04 BOOL  ; IND.MOV.MATERIAL
n95_05 95.05 BOOL  ; POSICION AUTO.SR
n95_06 95.06 BOOL  ; FALTA SR
n95_11 95.11 BOOL  ; AUX.REB.COLA A.I
n95_12 95.12 BOOL  ; AUX.REB.COLA B.I
n95_13 95.13 BOOL  ; AUX.REB.COLA A.D
n95_14 95.14 BOOL  ; AUX.REB.COLA B.D
n96_00 96.00 BOOL  ; PULSO MARCHA
n96_01 96.01 BOOL  ; AUX.PREMARCHA
n96_02 96.02 BOOL  ; MARCHA MAQU.EN B
n96_03 96.03 BOOL  ; AUX CLAXON PREMR
n96_04 96.04 BOOL  ; INIC.JOG.MAQUINA
n96_05 96.05 BOOL  ; AUX.JOG.MAQUINA
n96_06 96.06 BOOL  ; I.INI.CICLO GIRO
n96_07 96.07 BOOL  ; AUX.PRE-PARO
n96_08 96.08 BOOL  ; $?St$Bk?_#[981] / AUX.MODO "A"$?St$Bk?_#[981]
n96_09 96.09 BOOL  ; $?St$Bk?_#[982] / AUX.MODO "B"$?St$Bk?_#[982]
n96_10 96.10 BOOL  ; PARO EN FASE
n96_11 96.11 BOOL  ; CONDIC.MOD.B
n96_12 96.12 BOOL  ; I.IN MODO B
n96_13 96.13 BOOL  ; MARCH.ALARGADA
n96_14 96.14 BOOL  ; AUX.AVIS.PREPARO
n96_15 96.15 BOOL  ; AUX.PLT.PREPARO
n97_00 97.00 BOOL  ; I.DETECT.C/BOLS.
n97_02 97.02 BOOL  ; RESET PRESELEC.
n97_03 97.03 BOOL  ; COND.INIC.CICLO
n97_04 97.04 BOOL  ; PRESEL.ALCANZADA
n97_05 97.05 BOOL  ; INICIO CICLO
n97_06 97.06 BOOL  ; PRESEL.ERRONEA
n97_07 97.07 BOOL  ; I.AUX.TOTALZ.IZ.
n97_08 97.08 BOOL  ; I.AUX.TOTALZ.DR.
n97_11 97.11 BOOL  ; AUX.MAX.DIAMETRO
n97_12 97.12 BOOL  ; T.MAX.CICLO
n97_13 97.13 BOOL  ; I.INI.IMP.PRESEL
n97_14 97.14 BOOL  ; AUX.PLT.PRES.ERR
n97_15 97.15 BOOL  ; AUX.INIC.SOPLADO
n98_00 98.00 BOOL  ; EN CICLO
n98_01 98.01 BOOL  ; $?St$Bk?_#[983] / EN "1"$?St$Bk?_#[983]
n98_02 98.02 BOOL  ; $?St$Bk?_#[984] / EN "2"$?St$Bk?_#[984]
n98_03 98.03 BOOL  ; $?St$Bk?_#[985] / EN "3"$?St$Bk?_#[985]
n98_04 98.04 BOOL  ; $?St$Bk?_#[986] / EN "4"$?St$Bk?_#[986]
n98_05 98.05 BOOL  ; $?St$Bk?_#[987] / EN "5"$?St$Bk?_#[987]
n98_06 98.06 BOOL  ; $?St$Bk?_#[988] / EN "6"$?St$Bk?_#[988]
n98_07 98.07 BOOL  ; $?St$Bk?_#[989] / EN "7"$?St$Bk?_#[989]
n98_08 98.08 BOOL  ; $?St$Bk?_#[990] / EN "8"$?St$Bk?_#[990]
n98_09 98.09 BOOL  ; $?St$Bk?_#[991] / EN "9"$?St$Bk?_#[991]
n98_10 98.10 BOOL  ; FIN DE CICLO
n98_12 98.12 BOOL  ; AUX.EXTRACCION
n98_13 98.13 BOOL  ; DIAMETRO MAX.ACT
n98_14 98.14 BOOL  ; AUX.CLAX.DIAMTRO
n98_15 98.15 BOOL  ; IMP.DIAMETR.MAX
n99_01 99.01 BOOL  ; I.ABRIR PISONES
n99_05 99.05 BOOL  ; I.CIERR.PIS+SOPL
n99_06 99.06 BOOL  ; I.INTROD.MANDRIL
n99_08 99.08 BOOL  ; I.ABRIR SOPLADOR
n99_09 99.09 BOOL  ; I.EXTRAC.ROLLOS
n9_06 9.06 BOOL  ; ELV.GENERAL
nCNT143_PV C143 CHANNEL  ; MAX.CICLOS ASC.I
nCNT143_STATUS C0143 BOOL  ; MAX.CICLOS ASC.I
nCNT147_PV C147 CHANNEL  ; MAX.CICLOS.ASC.D
nCNT147_STATUS C0147 BOOL  ; MAX.CICLOS.ASC.D
nCNT176_PV C176 CHANNEL  ; ACTIV.EX/VOL.
nCNT176_STATUS C0176 BOOL  ; ACTIV.EX/VOL.
nCNT190_PV C190 CHANNEL  ; T.MONIT.CICLO
nCNT190_STATUS C0190 BOOL  ; T.MONIT.CICLO
nCNT217_PV C217 CHANNEL  ; RESET CONTADORES
nCNT217_STATUS C0217 BOOL  ; RESET CONTADORES
nCNT218_PV C218 CHANNEL  ; x5 DETEC.V.LIN.
nCNT218_STATUS C0218 BOOL  ; x5 DETEC.V.LIN.
nCNT220_PV C220 CHANNEL  ; 148M
nCNT220_STATUS C0220 BOOL  ; 148M
nCNT221_PV C221 CHANNEL  ; 138M
nCNT221_STATUS C0221 BOOL  ; 138M
nCNT222_PV C222 CHANNEL  ; 128M
nCNT222_STATUS C0222 BOOL  ; 128M
nCNT223_PV C223 CHANNEL  ; 120M
nCNT223_STATUS C0223 BOOL  ; 120M
nCNT224_PV C224 CHANNEL  ; 112M
nCNT224_STATUS C0224 BOOL  ; 112M
nCNT225_PV C225 CHANNEL  ; 104M
nCNT225_STATUS C0225 BOOL  ; 104M
nCNT226_PV C226 CHANNEL  ; 98M
nCNT226_STATUS C0226 BOOL  ; 98M
nCNT227_PV C227 CHANNEL  ; 91M
nCNT227_STATUS C0227 BOOL  ; 91M
nCNT228_PV C228 CHANNEL  ; 85M
nCNT228_STATUS C0228 BOOL  ; 85M
nCNT229_PV C229 CHANNEL  ; 79M
nCNT229_STATUS C0229 BOOL  ; 79M
nCNT230_PV C230 CHANNEL  ; 74M
nCNT230_STATUS C0230 BOOL  ; 74M
nCNT231_PV C231 CHANNEL  ; 69M
nCNT231_STATUS C0231 BOOL  ; 69M
nCNT232_PV C232 CHANNEL  ; 65M
nCNT232_STATUS C0232 BOOL  ; 65M
nCNT233_PV C233 CHANNEL  ; 60M
nCNT233_STATUS C0233 BOOL  ; 60M
nCNT234_PV C234 CHANNEL  ; 56M
nCNT234_STATUS C0234 BOOL  ; 56M
nCNT235_PV C235 CHANNEL  ; 52M
nCNT235_STATUS C0235 BOOL  ; 52M
nCNT236_PV C236 CHANNEL  ; 49M
nCNT236_STATUS C0236 BOOL  ; 49M
nCNT237_PV C237 CHANNEL  ; 46M
nCNT237_STATUS C0237 BOOL  ; 46M
nCNT238_PV C238 CHANNEL  ; 43M
nCNT238_STATUS C0238 BOOL  ; 43M
nCNT239_PV C239 CHANNEL  ; 40M
nCNT239_STATUS C0239 BOOL  ; 40M
nCNT240_PV C240 CHANNEL  ; 37M
nCNT240_STATUS C0240 BOOL  ; 37M
nCNT241_PV C241 CHANNEL  ; 35M
nCNT241_STATUS C0241 BOOL  ; 35M
nCNT242_PV C242 CHANNEL  ; 32M
nCNT242_STATUS C0242 BOOL  ; 32M
nCNT243_PV C243 CHANNEL  ; 30M
nCNT243_STATUS C0243 BOOL  ; 30M
nCNT244_PV C244 CHANNEL  ; 28M
nCNT244_STATUS C0244 BOOL  ; 28M
nCNT245_PV C245 CHANNEL  ; 26M
nCNT245_STATUS C0245 BOOL  ; 26M
nCNT246_PV C246 CHANNEL  ; 25M
nCNT246_STATUS C0246 BOOL  ; 25M
nCNT247_PV C247 CHANNEL  ; 23M
nCNT247_STATUS C0247 BOOL  ; 23M
nCNT248_PV C248 CHANNEL  ; 21M
nCNT248_STATUS C0248 BOOL  ; 21M
nCNT249_PV C249 CHANNEL  ; 20M
nCNT249_STATUS C0249 BOOL  ; 20M
nCNT261_PV C261 CHANNEL  ; PRESELECCION
nCNT261_STATUS C0261 BOOL  ; PRESELECCION
nCNT262_PV C262 CHANNEL  ; PRESELECTOR
nCNT262_STATUS C0262 BOOL  ; PRESELECTOR
nCNT265_PV C265 CHANNEL  ; ROLL.OPER.x1E0
nCNT265_STATUS C0265 BOOL  ; ROLL.OPER.x1E0
nCNT266_PV C266 CHANNEL  ; ROLL.OPER.x1E4
nCNT266_STATUS C0266 BOOL  ; ROLL.OPER.x1E4
nCNT270_PV C270 CHANNEL  ; GEN.1/10 HRS.
nCNT270_STATUS C0270 BOOL  ; GEN.1/10 HRS.
nCNT271_PV C271 CHANNEL  ; 1E-1 HORAS TRBJ.
nCNT271_STATUS C0271 BOOL  ; 1E-1 HORAS TRBJ.
nCNT272_PV C272 CHANNEL  ; 1E3 HRS.TRBJ.
nCNT272_STATUS C0272 BOOL  ; 1E3 HRS.TRBJ.
nCNT273_PV C273 CHANNEL  ; GEN 1/10 HRS.MAN
nCNT273_STATUS C0273 BOOL  ; GEN 1/10 HRS.MAN
nCNT274_PV C274 CHANNEL  ; 1E-1 HRS.MANIOBR
nCNT274_STATUS C0274 BOOL  ; 1E-1 HRS.MANIOBR
nCNT275_PV C275 CHANNEL  ; 1E3 HRS.MANIOBRA
nCNT275_STATUS C0275 BOOL  ; 1E3 HRS.MANIOBRA
nCNT280_PV C280 CHANNEL  ; PRESET.T.PRECAL
nCNT280_STATUS C0280 BOOL  ; PRESET.T.PRECAL
nCNT350_PV C350 CHANNEL  ; BASE DE TIEMPO
nCNT350_STATUS C0350 BOOL  ; BASE DE TIEMPO
nCNT84_PV C84 CHANNEL  ; AVIS.NO REGISTRO
nCNT84_STATUS C0084 BOOL  ; AVIS.NO REGISTRO
nHR0_06 H0.06 BOOL  ; SEL. I
nHR0_07 H0.07 BOOL  ; SEL. I+D
nHR0_08 H0.08 BOOL  ; SEL. D
nHR0_10 H0.10 BOOL  ; TECLA ENA.TOT.R.
nHR20_00 H20.00 BOOL  ; K.PISON IZD.
nHR20_01 H20.01 BOOL  ; K.PISON DRCH.
nHR20_02 H20.02 BOOL  ; K.BARRA SOPLADO
nHR20_03 H20.03 BOOL  ; K.EXTRACTOR IZD.
nHR20_04 H20.04 BOOL  ; K.EXTRACTOR DRCH
nHR20_05 H20.05 BOOL  ; K.VOLCADOR IZD.
nHR20_06 H20.06 BOOL  ; K.VOLCADOR DRCH.
nHR20_15 H20.15 BOOL  ; K.CAMBIO IDIOMA
nHR21_00 H21.00 BOOL  ; K.ASCENSOR IZD.
nHR21_01 H21.01 BOOL  ; K.ASCENSOR DRCH
nHR21_02 H21.02 BOOL  ; K.INTRODUCTOR IZ
nHR21_03 H21.03 BOOL  ; K.INTRODUCTOR DR
nHR21_05 H21.05 BOOL  ; K.IDA EXTRAC.IZ
nHR21_06 H21.06 BOOL  ; K.VUELT.EXTRAC.I
nHR21_07 H21.07 BOOL  ; K.IDA EXTRAC.DR
nHR21_08 H21.08 BOOL  ; K.VUELT.EXTRAC.D
nTIM0_PV T0 CHANNEL  ; T.PREDETERM.
nTIM0_STATUS T0000 BOOL  ; T.PREDETERM.
nTIM100_PV T100 CHANNEL  ; RETD.PREPOSICION
nTIM100_STATUS T0100 BOOL  ; RETD.PREPOSICION
nTIM101_PV T101 CHANNEL  ; RETD.G/MAN.TAMB.
nTIM101_STATUS T0101 BOOL  ; RETD.G/MAN.TAMB.
nTIM102_PV T102 CHANNEL  ; RETD.POSC.CILIND
nTIM102_STATUS T0102 BOOL  ; RETD.POSC.CILIND
nTIM103_PV T103 CHANNEL  ; T.MAX.CICLO
nTIM103_STATUS T0103 BOOL  ; T.MAX.CICLO
nTIM104_PV T104 CHANNEL  ; T.INIC.GIRO
nTIM104_STATUS T0104 BOOL  ; T.INIC.GIRO
nTIM109_PV T109 CHANNEL  ; RET.EXTRACCION
nTIM109_STATUS T0109 BOOL  ; RET.EXTRACCION
nTIM10_PV T10 CHANNEL  ; FRCUENC.AVIS.L.B
nTIM10_STATUS T0010 BOOL  ; FRCUENC.AVIS.L.B
nTIM110_PV T110 CHANNEL  ; T.ELV.PISON.I.A.
nTIM110_STATUS T0110 BOOL  ; T.ELV.PISON.I.A.
nTIM111_PV T111 CHANNEL  ; T.ELV.PISON D.A.
nTIM111_STATUS T0111 BOOL  ; T.ELV.PISON D.A.
nTIM112_PV T112 CHANNEL  ; T.ELV.VOLCD.I.C.
nTIM112_STATUS T0112 BOOL  ; T.ELV.VOLCD.I.C.
nTIM113_PV T113 CHANNEL  ; T.ELV.VOLCD.I.A.
nTIM113_STATUS T0113 BOOL  ; T.ELV.VOLCD.I.A.
nTIM114_PV T114 CHANNEL  ; T.ELV.VOLCD.D.C.
nTIM114_STATUS T0114 BOOL  ; T.ELV.VOLCD.D.C.
nTIM115_PV T115 CHANNEL  ; T.ELV.VOLCD.D.A.
nTIM115_STATUS T0115 BOOL  ; T.ELV.VOLCD.D.A.
nTIM116_PV T116 CHANNEL  ; T.ELV.ASCNS.I.A.
nTIM116_STATUS T0116 BOOL  ; T.ELV.ASCNS.I.A.
nTIM117_PV T117 CHANNEL  ; T.ELV.ASCNS.I.C.
nTIM117_STATUS T0117 BOOL  ; T.ELV.ASCNS.I.C.
nTIM118_PV T118 CHANNEL  ; T.ELV.ASCNS.D.A.
nTIM118_STATUS T0118 BOOL  ; T.ELV.ASCNS.D.A.
nTIM119_PV T119 CHANNEL  ; T.ELV.ASCNS.D.C.
nTIM119_STATUS T0119 BOOL  ; T.ELV.ASCNS.D.C.
nTIM11_PV T11 CHANNEL  ; T.AVIS.LOW BATT.
nTIM11_STATUS T0011 BOOL  ; T.AVIS.LOW BATT.
nTIM120_PV T120 CHANNEL  ; T.ELV.INTRD.I.C.
nTIM120_STATUS T0120 BOOL  ; T.ELV.INTRD.I.C.
nTIM121_PV T121 CHANNEL  ; T.ELV.INTRD.D.C.
nTIM121_STATUS T0121 BOOL  ; T.ELV.INTRD.D.C.
nTIM128_PV T128 CHANNEL  ; RTD.VOLCADOR I.
nTIM128_STATUS T0128 BOOL  ; RTD.VOLCADOR I.
nTIM129_PV T129 CHANNEL  ; RTD.VOLCADOR D.
nTIM129_STATUS T0129 BOOL  ; RTD.VOLCADOR D.
nTIM12_PV T12 CHANNEL  ; T.CLAXON LOW.BAT
nTIM12_STATUS T0012 BOOL  ; T.CLAXON LOW.BAT
nTIM130_PV T130 CHANNEL  ; RETD.RETOR.EXT.I
nTIM130_STATUS T0130 BOOL  ; RETD.RETOR.EXT.I
nTIM131_PV T131 CHANNEL  ; RETD.RET.EXTRC.D
nTIM131_STATUS T0131 BOOL  ; RETD.RET.EXTRC.D
nTIM132_PV T132 CHANNEL  ; RETD.ASC.LLENO I
nTIM132_STATUS T0132 BOOL  ; RETD.ASC.LLENO I
nTIM133_PV T133 CHANNEL  ; RETD.ASC.LLENO.D
nTIM133_STATUS T0133 BOOL  ; RETD.ASC.LLENO.D
nTIM134_PV T134 CHANNEL  ; RETD.RETR.MAND.I
nTIM134_STATUS T0134 BOOL  ; RETD.RETR.MAND.I
nTIM135_PV T135 CHANNEL  ; RETD.RETR.MAND.D
nTIM135_STATUS T0135 BOOL  ; RETD.RETR.MAND.D
nTIM136_PV T136 CHANNEL  ; RTD.DET.MANDR.I.
nTIM136_STATUS T0136 BOOL  ; RTD.DET.MANDR.I.
nTIM137_PV T137 CHANNEL  ; RTD.DET.MANDR.D.
nTIM137_STATUS T0137 BOOL  ; RTD.DET.MANDR.D.
nTIM140_PV T140 CHANNEL  ; RETD.SUB.ASC.IZD
nTIM140_STATUS T0140 BOOL  ; RETD.SUB.ASC.IZD
nTIM141_PV T141 CHANNEL  ; RETD.BAJ.ASC.IZD
nTIM141_STATUS T0141 BOOL  ; RETD.BAJ.ASC.IZD
nTIM142_PV T142 CHANNEL  ; RETD.INIC.ASC.IZ
nTIM142_STATUS T0142 BOOL  ; RETD.INIC.ASC.IZ
nTIM144_PV T144 CHANNEL  ; RETD.SUB.ASC.DRH
nTIM144_STATUS T0144 BOOL  ; RETD.SUB.ASC.DRH
nTIM145_PV T145 CHANNEL  ; RETD.BAJ.ASC.DRH
nTIM145_STATUS T0145 BOOL  ; RETD.BAJ.ASC.DRH
nTIM146_PV T146 CHANNEL  ; RETD.INIC.ASC.DR
nTIM146_STATUS T0146 BOOL  ; RETD.INIC.ASC.DR
nTIM148_PV T148 CHANNEL  ; RETD.AVIS.DEPOSI
nTIM148_STATUS T0148 BOOL  ; RETD.AVIS.DEPOSI
nTIM15_PV T15 CHANNEL  ; RETD.FI.DETC.GIR
nTIM15_STATUS T0015 BOOL  ; RETD.FI.DETC.GIR
nTIM160_PV T160 CHANNEL  ; RETD.VOLC.VACIOS
nTIM160_STATUS T0160 BOOL  ; RETD.VOLC.VACIOS
nTIM161_PV T161 CHANNEL  ; RETD.CONDIC.GIRO
nTIM161_STATUS T0161 BOOL  ; RETD.CONDIC.GIRO
nTIM162_PV T162 CHANNEL  ; $?St$Bk?_#[992] / PAUSA CICLO "A"$?St$Bk?_#[992]
nTIM162_STATUS T0162 BOOL  ; $?St$Bk?_#[993] / PAUSA CICLO "A"$?St$Bk?_#[993]
nTIM163_PV T163 CHANNEL  ; RETD.COND.GIR.B
nTIM163_STATUS T0163 BOOL  ; RETD.COND.GIR.B
nTIM164_PV T164 CHANNEL  ; LIMITE INIC.GIRO
nTIM164_STATUS T0164 BOOL  ; LIMITE INIC.GIRO
nTIM166_PV T166 CHANNEL  ; T.AVIS.POSIC.C3
nTIM166_STATUS T0166 BOOL  ; T.AVIS.POSIC.C3
nTIM167_PV T167 CHANNEL  ; T.PARO POSICION
nTIM167_STATUS T0167 BOOL  ; T.PARO POSICION
nTIM168_PV T168 CHANNEL  ; RESET INTEGRADOR
nTIM168_STATUS T0168 BOOL  ; RESET INTEGRADOR
nTIM169_PV T169 CHANNEL  ; RETARD.PARO REBO
nTIM169_STATUS T0169 BOOL  ; RETARD.PARO REBO
nTIM170_PV T170 CHANNEL  ; T.FRENO A.IZD.
nTIM170_STATUS T0170 BOOL  ; T.FRENO A.IZD.
nTIM171_PV T171 CHANNEL  ; T.FRENO B.IZD.
nTIM171_STATUS T0171 BOOL  ; T.FRENO B.IZD.
nTIM172_PV T172 CHANNEL  ; T.FRENO A.DRCH.
nTIM172_STATUS T0172 BOOL  ; T.FRENO A.DRCH.
nTIM173_PV T173 CHANNEL  ; T.FRENO B.DRCH
nTIM173_STATUS T0173 BOOL  ; T.FRENO B.DRCH
nTIM1_PV T1 CHANNEL  ; CAMBIO IDIOMA
nTIM1_STATUS T0001 BOOL  ; CAMBIO IDIOMA
nTIM200_PV T200 CHANNEL  ; RET.MLF.STOPS
nTIM200_STATUS T0200 BOOL  ; RET.MLF.STOPS
nTIM201_PV T201 CHANNEL  ; T.PERMIS.RESET
nTIM201_STATUS T0201 BOOL  ; T.PERMIS.RESET
nTIM202_PV T202 CHANNEL  ; TIM.INI.REARME
nTIM202_STATUS T0202 BOOL  ; TIM.INI.REARME
nTIM203_PV T203 CHANNEL  ; TIM.FIN REARME
nTIM203_STATUS T0203 BOOL  ; TIM.FIN REARME
nTIM204_PV T204 CHANNEL  ; TIM.SUBIDA AIRE
nTIM204_STATUS T0204 BOOL  ; TIM.SUBIDA AIRE
nTIM205_PV T205 CHANNEL  ; TIM.AIRE O.K.
nTIM205_STATUS T0205 BOOL  ; TIM.AIRE O.K.
nTIM206_PV T206 CHANNEL  ; TIM.MLF.MICR.PRT
nTIM206_STATUS T0206 BOOL  ; TIM.MLF.MICR.PRT
nTIM207_PV T207 CHANNEL  ; TIM.AUTORRESTART
nTIM207_STATUS T0207 BOOL  ; TIM.AUTORRESTART
nTIM208_PV T208 CHANNEL  ; TIM.MSG.PRTA.TMB
nTIM208_STATUS T0208 BOOL  ; TIM.MSG.PRTA.TMB
nTIM209_PV T209 CHANNEL  ; TIM.MLF.CIRC.PUE
nTIM209_STATUS T0209 BOOL  ; TIM.MLF.CIRC.PUE
nTIM210_PV T210 CHANNEL  ; TIM.ESPERA AIRE2
nTIM210_STATUS T0210 BOOL  ; TIM.ESPERA AIRE2
nTIM211_PV T211 CHANNEL  ; T.REB.COLA A.I.
nTIM211_STATUS T0211 BOOL  ; T.REB.COLA A.I.
nTIM212_PV T212 CHANNEL  ; T.REB.COLA B.I.
nTIM212_STATUS T0212 BOOL  ; T.REB.COLA B.I.
nTIM213_PV T213 CHANNEL  ; T.REB.COLA A.D.
nTIM213_STATUS T0213 BOOL  ; T.REB.COLA A.D.
nTIM214_PV T214 CHANNEL  ; T.REB.COLA B.D.
nTIM214_STATUS T0214 BOOL  ; T.REB.COLA B.D.
nTIM219_PV T219 CHANNEL  ; SELEC.LEVA CLK 2
nTIM219_STATUS T0219 BOOL  ; SELEC.LEVA CLK 2
nTIM260_PV T260 CHANNEL  ; T.AUTORREPEAT
nTIM260_STATUS T0260 BOOL  ; T.AUTORREPEAT
nTIM267_PV T267 CHANNEL  ; RET.RST.TOT.RLLS
nTIM267_STATUS T0267 BOOL  ; RET.RST.TOT.RLLS
nTIM26_PV T26 CHANNEL  ; T.CAX.TAMBOR
nTIM26_STATUS T0026 BOOL  ; T.CAX.TAMBOR
nTIM27_PV T27 CHANNEL  ; T.CAX.VIBRAD.IZ.
nTIM27_STATUS T0027 BOOL  ; T.CAX.VIBRAD.IZ.
nTIM281_PV T281 CHANNEL  ; T.PRECAL.
nTIM281_STATUS T0281 BOOL  ; T.PRECAL.
nTIM28_PV T28 CHANNEL  ; T.CAX.VIBRAD.DR.
nTIM28_STATUS T0028 BOOL  ; T.CAX.VIBRAD.DR.
nTIM299_PV T299 CHANNEL  ; T.KEEP JMP.SUBRT
nTIM299_STATUS T0299 BOOL  ; T.KEEP JMP.SUBRT
nTIM300_PV T300 CHANNEL  ; TH.PI.
nTIM300_STATUS T0300 BOOL  ; TH.PI.
nTIM301_PV T301 CHANNEL  ; THS.PSN
nTIM301_STATUS T0301 BOOL  ; THS.PSN
nTIM302_PV T302 CHANNEL  ; THL.PSN
nTIM302_STATUS T0302 BOOL  ; THL.PSN
nTIM303_PV T303 CHANNEL  ; TH.CERRAR PSN
nTIM303_STATUS T0303 BOOL  ; TH.CERRAR PSN
nTIM304_PV T304 CHANNEL  ; THS.CERR.EXTRAC
nTIM304_STATUS T0304 BOOL  ; THS.CERR.EXTRAC
nTIM305_PV T305 CHANNEL  ; THL.CERR.EXTRAC
nTIM305_STATUS T0305 BOOL  ; THL.CERR.EXTRAC
nTIM306_PV T306 CHANNEL  ; THS.ABRIR EXTRCT
nTIM306_STATUS T0306 BOOL  ; THS.ABRIR EXTRCT
nTIM307_PV T307 CHANNEL  ; THL.ABRIR EXTRAT
nTIM307_STATUS T0307 BOOL  ; THL.ABRIR EXTRAT
nTIM308_PV T308 CHANNEL  ; THS.ABRIR INTRO
nTIM308_STATUS T0308 BOOL  ; THS.ABRIR INTRO
nTIM309_PV T309 CHANNEL  ; THL.ABRIR INTRO
nTIM309_STATUS T0309 BOOL  ; THL.ABRIR INTRO
nTIM310_PV T310 CHANNEL  ; THS.ABRIR SOPLAD
nTIM310_STATUS T0310 BOOL  ; THS.ABRIR SOPLAD
nTIM311_PV T311 CHANNEL  ; THL.ABRIR SOPLAD
nTIM311_STATUS T0311 BOOL  ; THL.ABRIR SOPLAD
nTIM312_PV T312 CHANNEL  ; THS.CERR.SOPLAD
nTIM312_STATUS T0312 BOOL  ; THS.CERR.SOPLAD
nTIM313_PV T313 CHANNEL  ; THL.CERR.SOPLADO
nTIM313_STATUS T0313 BOOL  ; THL.CERR.SOPLADO
nTIM314_PV T314 CHANNEL  ; TS.PRESOSTATO
nTIM314_STATUS T0314 BOOL  ; TS.PRESOSTATO
nTIM315_PV T315 CHANNEL  ; TL.PRESOSTATO
nTIM315_STATUS T0315 BOOL  ; TL.PRESOSTATO
nTIM316_PV T316 CHANNEL  ; T.AJUSTE PRESOST
nTIM316_STATUS T0316 BOOL  ; T.AJUSTE PRESOST
nTIM317_PV T317 CHANNEL  ; T.PITO.PRESOSTAT
nTIM317_STATUS T0317 BOOL  ; T.PITO.PRESOSTAT
nTIM320_PV T320 CHANNEL  ; CONTROL SOPLADRS
nTIM320_STATUS T0320 BOOL  ; CONTROL SOPLADRS
nTIM321_PV T321 CHANNEL  ; ABR/CERR.SOPLADR
nTIM321_STATUS T0321 BOOL  ; ABR/CERR.SOPLADR
nTIM330_PV T330 CHANNEL  ; T.2PI
nTIM330_STATUS T0330 BOOL  ; T.2PI
nTIM331_PV T331 CHANNEL  ; T.PREDETERM.
nTIM331_STATUS T0331 BOOL  ; T.PREDETERM.
nTIM33_PV T33 CHANNEL  ; RETD.FIN BOBINA
nTIM33_STATUS T0033 BOOL  ; RETD.FIN BOBINA
nTIM34_PV T34 CHANNEL  ; FREC.AVIS FI.BOB
nTIM34_STATUS T0034 BOOL  ; FREC.AVIS FI.BOB
nTIM35_PV T35 CHANNEL  ; DURAC.AVIS.FI.BO
nTIM35_STATUS T0035 BOOL  ; DURAC.AVIS.FI.BO
nTIM360_PV T360 CHANNEL  ; T.L.V.CEL.3505
nTIM360_STATUS T0360 BOOL  ; T.L.V.CEL.3505
nTIM361_PV T361 CHANNEL  ; T.S.V.CEL.3505
nTIM361_STATUS T0361 BOOL  ; T.S.V.CEL.3505
nTIM362_PV T362 CHANNEL  ; T.L.V.CEL.3506
nTIM362_STATUS T0362 BOOL  ; T.L.V.CEL.3506
nTIM363_PV T363 CHANNEL  ; T.S.V.CEL.3506
nTIM363_STATUS T0363 BOOL  ; T.S.V.CEL.3506
nTIM364_PV T364 CHANNEL  ; T.L.V.CEL.3605
nTIM364_STATUS T0364 BOOL  ; T.L.V.CEL.3605
nTIM365_PV T365 CHANNEL  ; T.S.V.CEL.3605
nTIM365_STATUS T0365 BOOL  ; T.S.V.CEL.3605
nTIM366_PV T366 CHANNEL  ; T.L.V.CEL.3606
nTIM366_STATUS T0366 BOOL  ; T.L.V.CEL.3606
nTIM367_PV T367 CHANNEL  ; T.S.V.CEL.3606
nTIM367_STATUS T0367 BOOL  ; T.S.V.CEL.3606
nTIM368_PV T368 CHANNEL  ; T.L.V.CEL.3700
nTIM368_STATUS T0368 BOOL  ; T.L.V.CEL.3700
nTIM369_PV T369 CHANNEL  ; T.S.V.CEL.3700
nTIM369_STATUS T0369 BOOL  ; T.S.V.CEL.3700
nTIM36_PV T36 CHANNEL  ; AVIS.TOT.FI.BOBI
nTIM36_STATUS T0036 BOOL  ; AVIS.TOT.FI.BOBI
nTIM370_PV T370 CHANNEL  ; T.L.V.CEL.3701
nTIM370_STATUS T0370 BOOL  ; T.L.V.CEL.3701
nTIM371_PV T371 CHANNEL  ; T.S.V.CEL.3701
nTIM371_STATUS T0371 BOOL  ; T.S.V.CEL.3701
nTIM372_PV T372 CHANNEL  ; T.L.V.CEL.3705
nTIM372_STATUS T0372 BOOL  ; T.L.V.CEL.3705
nTIM373_PV T373 CHANNEL  ; T.S.V.CEL.3705
nTIM373_STATUS T0373 BOOL  ; T.S.V.CEL.3705
nTIM374_PV T374 CHANNEL  ; T.L.V.CEL.3708
nTIM374_STATUS T0374 BOOL  ; T.L.V.CEL.3708
nTIM375_PV T375 CHANNEL  ; T.S.V.CEL.3708
nTIM375_STATUS T0375 BOOL  ; T.S.V.CEL.3708
nTIM376_PV T376 CHANNEL  ; T.L.V.CEL.3709
nTIM376_STATUS T0376 BOOL  ; T.L.V.CEL.3709
nTIM377_PV T377 CHANNEL  ; T.S.V.CEL.3709
nTIM377_STATUS T0377 BOOL  ; T.S.V.CEL.3709
nTIM378_PV T378 CHANNEL  ; T.L.V.CEL.3713
nTIM378_STATUS T0378 BOOL  ; T.L.V.CEL.3713
nTIM379_PV T379 CHANNEL  ; T.S.V.CEL.3713
nTIM379_STATUS T0379 BOOL  ; T.S.V.CEL.3713
nTIM37_PV T37 CHANNEL  ; T.MSG. FI BOBINA
nTIM37_STATUS T0037 BOOL  ; T.MSG. FI BOBINA
nTIM380_PV T380 CHANNEL  ; TH.PITOS CEL
nTIM380_STATUS T0380 BOOL  ; TH.PITOS CEL
nTIM3_PV T3 CHANNEL  ; TH.DURACC.SOPLAD
nTIM3_STATUS T0003 BOOL  ; TH.DURACC.SOPLAD
nTIM45_PV T45 CHANNEL  ; T.AVIS.DIAMT.MAX
nTIM45_STATUS T0045 BOOL  ; T.AVIS.DIAMT.MAX
nTIM4_PV T4 CHANNEL  ; TH RETD.C/VELO.
nTIM4_STATUS T0004 BOOL  ; TH RETD.C/VELO.
nTIM50_PV T50 CHANNEL  ; T.RESET
nTIM50_STATUS T0050 BOOL  ; T.RESET
nTIM52_PV T52 CHANNEL  ; RETARD.V.LENT.MW
nTIM52_STATUS T0052 BOOL  ; RETARD.V.LENT.MW
nTIM55_PV T55 CHANNEL  ; RETAD.ALRM.T.SR.
nTIM55_STATUS T0055 BOOL  ; RETAD.ALRM.T.SR.
nTIM56_PV T56 CHANNEL  ; T.RETD.PREMARCHA
nTIM56_STATUS T0056 BOOL  ; T.RETD.PREMARCHA
nTIM57_PV T57 CHANNEL  ; PITO CLX.PREMARC
nTIM57_STATUS T0057 BOOL  ; PITO CLX.PREMARC
nTIM58_PV T58 CHANNEL  ; PAUSA CLX.PREMAR
nTIM58_STATUS T0058 BOOL  ; PAUSA CLX.PREMAR
nTIM59_PV T59 CHANNEL  ; RETD.JOG.MAQUINA
nTIM59_STATUS T0059 BOOL  ; RETD.JOG.MAQUINA
nTIM5_PV T5 CHANNEL  ; TH.RETD.SOPLADO
nTIM5_STATUS T0005 BOOL  ; TH.RETD.SOPLADO
nTIM60_PV T60 CHANNEL  ; RETD.FIN MOV.MAT
nTIM60_STATUS T0060 BOOL  ; RETD.FIN MOV.MAT
nTIM61_PV T61 CHANNEL  ; ALARGA MARCHA
nTIM61_STATUS T0061 BOOL  ; ALARGA MARCHA
nTIM63_PV T63 CHANNEL  ; MULT.x2 TOTALIZD
nTIM63_STATUS T0063 BOOL  ; MULT.x2 TOTALIZD
nTIM67_PV T67 CHANNEL  ; RETD.INI.ZIGZAG
nTIM67_STATUS T0067 BOOL  ; RETD.INI.ZIGZAG
nTIM70_PV T70 CHANNEL  ; T.DET.R.CAIDO IZ
nTIM70_STATUS T0070 BOOL  ; T.DET.R.CAIDO IZ
nTIM71_PV T71 CHANNEL  ; T.DET.R.CAIDO DR
nTIM71_STATUS T0071 BOOL  ; T.DET.R.CAIDO DR
nTIM72_PV T72 CHANNEL  ; T.AVIS.R.CAID.IZ
nTIM72_STATUS T0072 BOOL  ; T.AVIS.R.CAID.IZ
nTIM73_PV T73 CHANNEL  ; T.AVIS.R.CAID.DR
nTIM73_STATUS T0073 BOOL  ; T.AVIS.R.CAID.DR
nTIM74_PV T74 CHANNEL  ; RET.EXTRACCION
nTIM74_STATUS T0074 BOOL  ; RET.EXTRACCION
nTIM80_PV T80 CHANNEL  ; RET.MSG.38
nTIM80_STATUS T0080 BOOL  ; RET.MSG.38
nTIM83_PV T83 CHANNEL  ; RET.AVIS.NO REGS
nTIM83_STATUS T0083 BOOL  ; RET.AVIS.NO REGS
nTIM90_PV T90 CHANNEL  ; MESG.EXTR.IZD.
nTIM90_STATUS T0090 BOOL  ; MESG.EXTR.IZD.
nTIM91_PV T91 CHANNEL  ; MSG.EXTRAC.DRCH.
nTIM91_STATUS T0091 BOOL  ; MSG.EXTRAC.DRCH.
nTIM96_PV T96 CHANNEL  ; T.AVIS.PREPARO
nTIM96_STATUS T0096 BOOL  ; T.AVIS.PREPARO

## Program MainProgram (cyclic task 0)

### Section ConfigAnalogiques

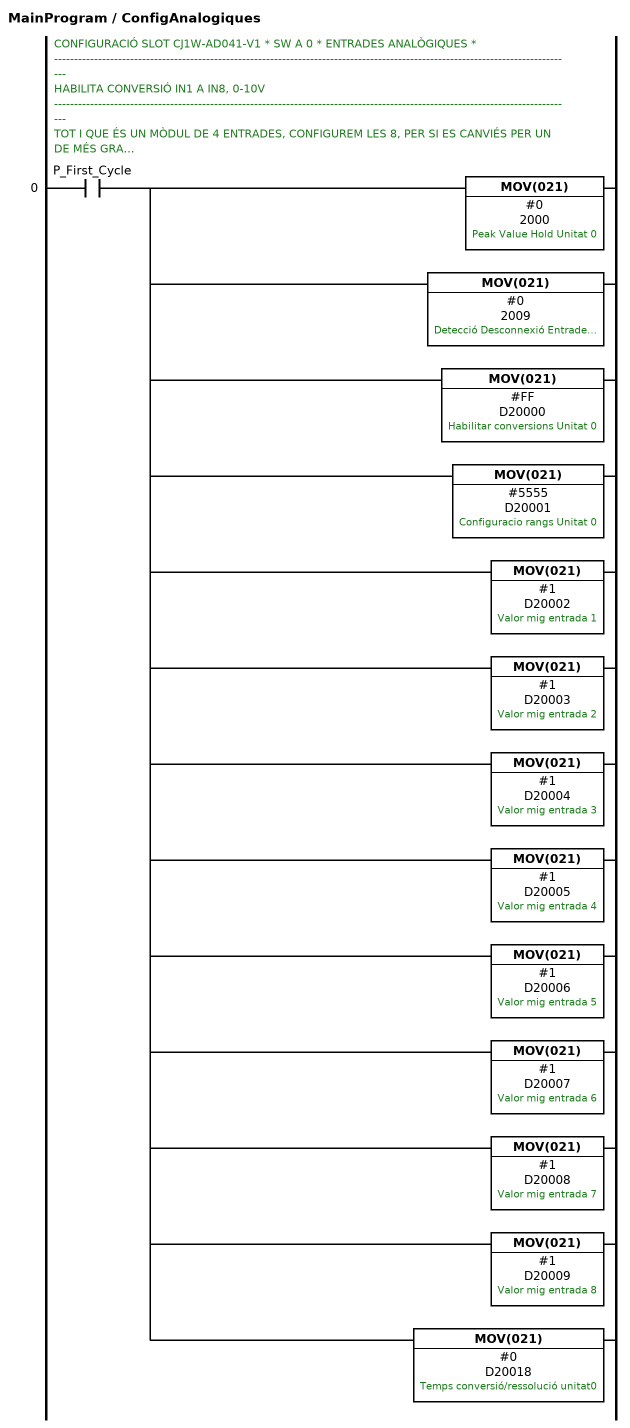
; rung 0: CONFIGURACIÓ SLOT CJ1W-AD041-V1 * SW A 0 * ENTRADES ANALÒGIQUES * / ---------------------------------------------------------------------------------------------------------------------------------- / HABILITA CONVERSIÓ IN1 A IN8, 0-10V / ---------------------------------------------------------------------------------------------------------------------------------- / TOT I QUE ÉS UN MÒDUL DE 4 ENTRADES, CONFIGUREM LES 8, PER SI ES CANVIÉS PER UN DE MÉS GRAN / ----------------------------------------------------------------------------------------------------------------------------------
LD P_First_Cycle
MOV(021) #0 2000  ; Peak Value Hold Unitat 0
MOV(021) #0 2009  ; Detecció Desconnexió Entrades Unitat 0
MOV(021) #FF D20000  ; Habilitar conversions Unitat 0
MOV(021) #5555 D20001  ; Configuracio rangs Unitat 0
MOV(021) #1 D20002  ; Valor mig entrada 1
MOV(021) #1 D20003  ; Valor mig entrada 2
MOV(021) #1 D20004  ; Valor mig entrada 3
MOV(021) #1 D20005  ; Valor mig entrada 4
MOV(021) #1 D20006  ; Valor mig entrada 5
MOV(021) #1 D20007  ; Valor mig entrada 6
MOV(021) #1 D20008  ; Valor mig entrada 7
MOV(021) #1 D20009  ; Valor mig entrada 8
MOV(021) #0 D20018  ; Temps conversió/ressolució unitat0

### Section Inicialitzacions

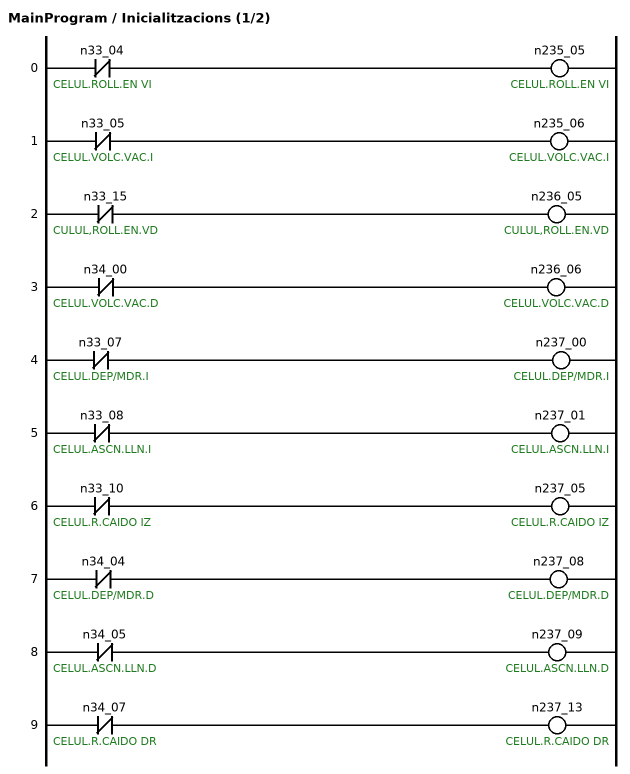
; rung 0
LDNOT n33_04  ; CELUL.ROLL.EN VI
OUT n235_05  ; CELUL.ROLL.EN VI
; rung 1
LDNOT n33_05  ; CELUL.VOLC.VAC.I
OUT n235_06  ; CELUL.VOLC.VAC.I
; rung 2
LDNOT n33_15  ; CULUL,ROLL.EN.VD
OUT n236_05  ; CULUL,ROLL.EN.VD
; rung 3
LDNOT n34_00  ; CELUL.VOLC.VAC.D
OUT n236_06  ; CELUL.VOLC.VAC.D
; rung 4
LDNOT n33_07  ; CELUL.DEP/MDR.I
OUT n237_00  ; CELUL.DEP/MDR.I
; rung 5
LDNOT n33_08  ; CELUL.ASCN.LLN.I
OUT n237_01  ; CELUL.ASCN.LLN.I
; rung 6
LDNOT n33_10  ; CELUL.R.CAIDO IZ
OUT n237_05  ; CELUL.R.CAIDO IZ
; rung 7
LDNOT n34_04  ; CELUL.DEP/MDR.D
OUT n237_08  ; CELUL.DEP/MDR.D
; rung 8
LDNOT n34_05  ; CELUL.ASCN.LLN.D
OUT n237_09  ; CELUL.ASCN.LLN.D
; rung 9
LDNOT n34_07  ; CELUL.R.CAIDO DR
OUT n237_13  ; CELUL.R.CAIDO DR

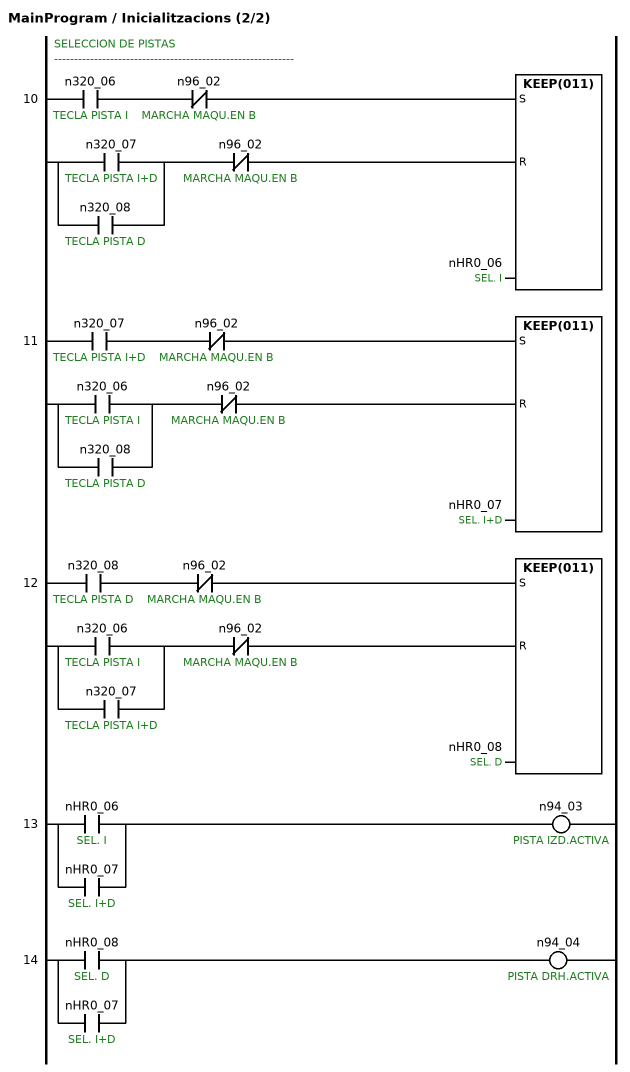
; rung 10: SELECCION DE PISTAS / ------------------------------------------------------------
LD n320_06  ; TECLA PISTA I
ANDNOT n96_02  ; MARCHA MAQU.EN B
LD n320_07  ; TECLA PISTA I+D
OR n320_08  ; TECLA PISTA D
ANDNOT n96_02  ; MARCHA MAQU.EN B
KEEP(011) nHR0_06  ; SEL. I
; rung 11
LD n320_07  ; TECLA PISTA I+D
ANDNOT n96_02  ; MARCHA MAQU.EN B
LD n320_06  ; TECLA PISTA I
OR n320_08  ; TECLA PISTA D
ANDNOT n96_02  ; MARCHA MAQU.EN B
KEEP(011) nHR0_07  ; SEL. I+D
; rung 12
LD n320_08  ; TECLA PISTA D
ANDNOT n96_02  ; MARCHA MAQU.EN B
LD n320_06  ; TECLA PISTA I
OR n320_07  ; TECLA PISTA I+D
ANDNOT n96_02  ; MARCHA MAQU.EN B
KEEP(011) nHR0_08  ; SEL. D
; rung 13
LD nHR0_06  ; SEL. I
OR nHR0_07  ; SEL. I+D
OUT n94_03  ; PISTA IZD.ACTIVA
; rung 14
LD nHR0_08  ; SEL. D
OR nHR0_07  ; SEL. I+D
OUT n94_04  ; PISTA DRH.ACTIVA

### Section Emergencies

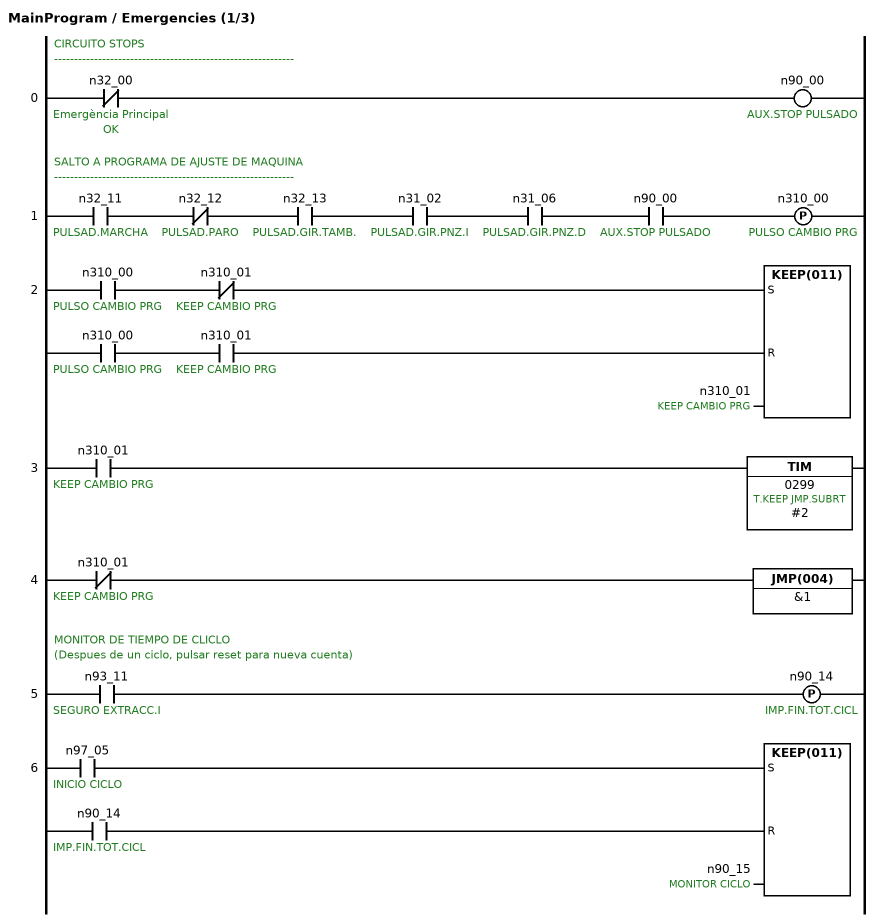
; rung 0: CIRCUITO STOPS / ------------------------------------------------------------
LDNOT n32_00  ; Emergència Principal OK
OUT n90_00  ; AUX.STOP PULSADO
; rung 1: SALTO A PROGRAMA DE AJUSTE DE MAQUINA / ------------------------------------------------------------
LD n32_11  ; PULSAD.MARCHA
ANDNOT n32_12  ; PULSAD.PARO
AND n32_13  ; PULSAD.GIR.TAMB.
AND n31_02  ; PULSAD.GIR.PNZ.I
AND n31_06  ; PULSAD.GIR.PNZ.D
AND n90_00  ; AUX.STOP PULSADO
DIFU(013) n310_00  ; PULSO CAMBIO PRG
; rung 2
LD n310_00  ; PULSO CAMBIO PRG
ANDNOT n310_01  ; KEEP CAMBIO PRG
LD n310_00  ; PULSO CAMBIO PRG
AND n310_01  ; KEEP CAMBIO PRG
KEEP(011) n310_01  ; KEEP CAMBIO PRG
; rung 3
LD n310_01  ; KEEP CAMBIO PRG
TIM 0299 #2  ; T.KEEP JMP.SUBRT
; rung 4
LDNOT n310_01  ; KEEP CAMBIO PRG
JMP(004) &1
; rung 5: MONITOR DE TIEMPO DE CLICLO / (Despues de un ciclo, pulsar reset para nueva cuenta)
LD n93_11  ; SEGURO EXTRACC.I
DIFU(013) n90_14  ; IMP.FIN.TOT.CICL
; rung 6
LD n97_05  ; INICIO CICLO
LD n90_14  ; IMP.FIN.TOT.CICL
KEEP(011) n90_15  ; MONITOR CICLO

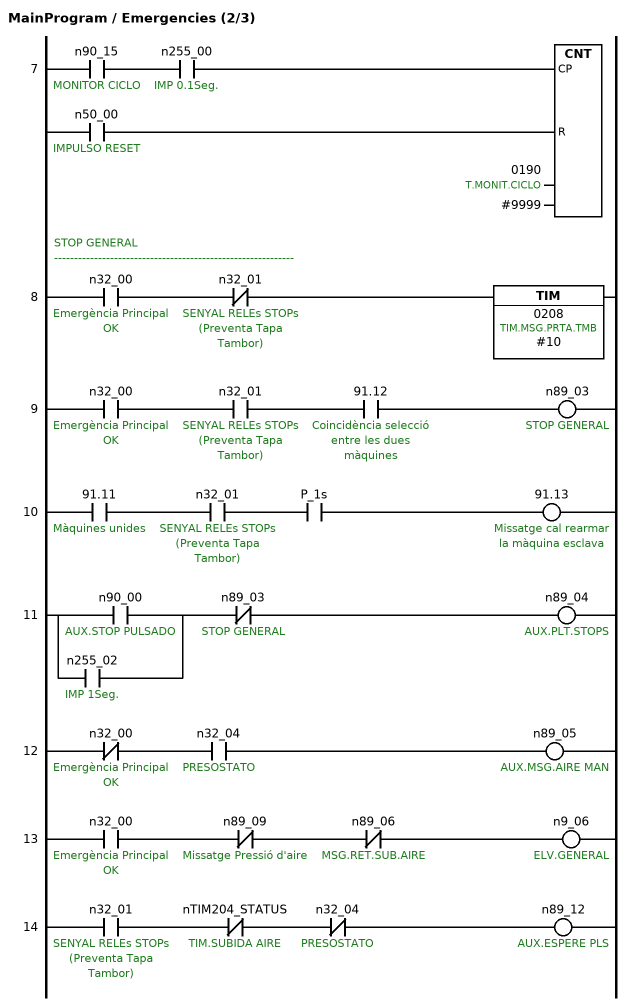
; rung 7
LD n90_15  ; MONITOR CICLO
AND n255_00  ; IMP 0.1Seg.
LD n50_00  ; IMPULSO RESET
CNT 0190 #9999  ; T.MONIT.CICLO
; rung 8: STOP GENERAL / ------------------------------------------------------------
LD n32_00  ; Emergència Principal OK
ANDNOT n32_01  ; SENYAL RELEs STOPs (Preventa Tapa Tambor)
TIM 0208 #10  ; TIM.MSG.PRTA.TMB
; rung 9
LD n32_00  ; Emergència Principal OK
AND n32_01  ; SENYAL RELEs STOPs (Preventa Tapa Tambor)
AND 91.12  ; Coincidència selecció entre les dues màquines
OUT n89_03  ; STOP GENERAL
; rung 10
LD 91.11  ; Màquines unides
AND n32_01  ; SENYAL RELEs STOPs (Preventa Tapa Tambor)
AND P_1s
OUT 91.13  ; Missatge cal rearmar la màquina esclava
; rung 11
LD n90_00  ; AUX.STOP PULSADO
OR n255_02  ; IMP 1Seg.
ANDNOT n89_03  ; STOP GENERAL
OUT n89_04  ; AUX.PLT.STOPS
; rung 12
LDNOT n32_00  ; Emergència Principal OK
AND n32_04  ; PRESOSTATO
OUT n89_05  ; AUX.MSG.AIRE MAN
; rung 13
LD n32_00  ; Emergència Principal OK
ANDNOT n89_09  ; Missatge Pressió d'aire
ANDNOT n89_06  ; MSG.RET.SUB.AIRE
OUT n9_06  ; ELV.GENERAL
; rung 14
LD n32_01  ; SENYAL RELEs STOPs (Preventa Tapa Tambor)
ANDNOT nTIM204_STATUS  ; TIM.SUBIDA AIRE
ANDNOT n32_04  ; PRESOSTATO
OUT n89_12  ; AUX.ESPERE PLS

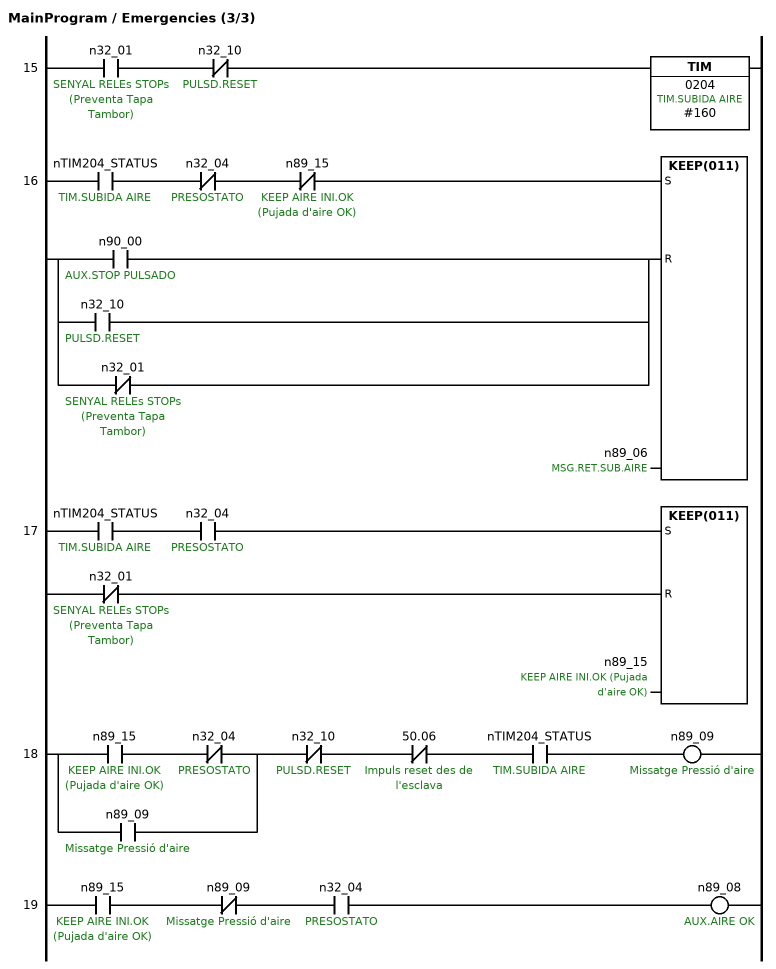
; rung 15
LD n32_01  ; SENYAL RELEs STOPs (Preventa Tapa Tambor)
ANDNOT n32_10  ; PULSD.RESET
TIM 0204 #160  ; TIM.SUBIDA AIRE
; rung 16
LD nTIM204_STATUS  ; TIM.SUBIDA AIRE
ANDNOT n32_04  ; PRESOSTATO
ANDNOT n89_15  ; KEEP AIRE INI.OK (Pujada d'aire OK)
LD n90_00  ; AUX.STOP PULSADO
OR n32_10  ; PULSD.RESET
ORNOT n32_01  ; SENYAL RELEs STOPs (Preventa Tapa Tambor)
KEEP(011) n89_06  ; MSG.RET.SUB.AIRE
; rung 17
LD nTIM204_STATUS  ; TIM.SUBIDA AIRE
AND n32_04  ; PRESOSTATO
LDNOT n32_01  ; SENYAL RELEs STOPs (Preventa Tapa Tambor)
KEEP(011) n89_15  ; KEEP AIRE INI.OK (Pujada d'aire OK)
; rung 18
LD n89_15  ; KEEP AIRE INI.OK (Pujada d'aire OK)
ANDNOT n32_04  ; PRESOSTATO
OR n89_09  ; Missatge Pressió d'aire
ANDNOT n32_10  ; PULSD.RESET
ANDNOT 50.06  ; Impuls reset des de l'esclava
AND nTIM204_STATUS  ; TIM.SUBIDA AIRE
OUT n89_09  ; Missatge Pressió d'aire
; rung 19
LD n89_15  ; KEEP AIRE INI.OK (Pujada d'aire OK)
ANDNOT n89_09  ; Missatge Pressió d'aire
AND n32_04  ; PRESOSTATO
OUT n89_08  ; AUX.AIRE OK

### Section maquina

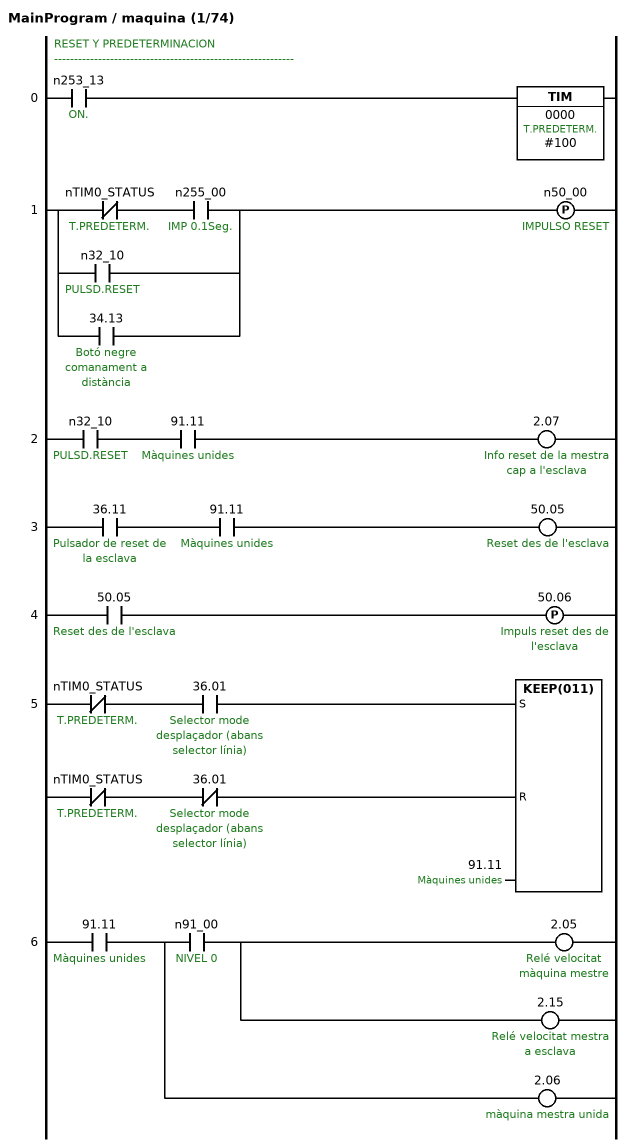
; rung 0: RESET Y PREDETERMINACION / ------------------------------------------------------------
LD n253_13  ; ON.
TIM 0000 #100  ; T.PREDETERM.
; rung 1
LDNOT nTIM0_STATUS  ; T.PREDETERM.
AND n255_00  ; IMP 0.1Seg.
OR n32_10  ; PULSD.RESET
OR 34.13  ; Botó negre comanament a distància
DIFU(013) n50_00  ; IMPULSO RESET
; rung 2
LD n32_10  ; PULSD.RESET
AND 91.11  ; Màquines unides
OUT 2.07  ; Info reset de la mestra cap a l'esclava
; rung 3
LD 36.11  ; Pulsador de reset de la esclava
AND 91.11  ; Màquines unides
OUT 50.05  ; Reset des de l'esclava
; rung 4
LD 50.05  ; Reset des de l'esclava
DIFU(013) 50.06  ; Impuls reset des de l'esclava
; rung 5
LDNOT nTIM0_STATUS  ; T.PREDETERM.
AND 36.01  ; Selector mode desplaçador (abans selector línia)
LDNOT nTIM0_STATUS  ; T.PREDETERM.
ANDNOT 36.01  ; Selector mode desplaçador (abans selector línia)
KEEP(011) 91.11  ; Màquines unides
; rung 6
LD 91.11  ; Màquines unides
OUT TR0
AND n91_00  ; NIVEL 0
OUT 2.05  ; Relé velocitat màquina mestre
OUT 2.15  ; Relé velocitat mestra a esclava
LD TR0
OUT 2.06  ; màquina mestra unida

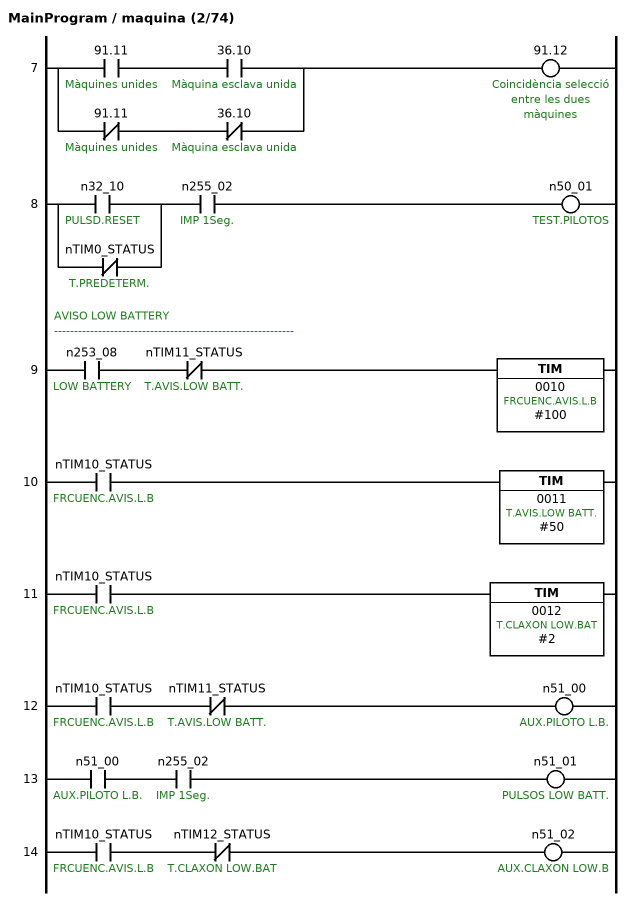
; rung 7
LD 91.11  ; Màquines unides
AND 36.10  ; Màquina esclava unida
LDNOT 91.11  ; Màquines unides
ANDNOT 36.10  ; Màquina esclava unida
ORLD
OUT 91.12  ; Coincidència selecció entre les dues màquines
; rung 8
LD n32_10  ; PULSD.RESET
ORNOT nTIM0_STATUS  ; T.PREDETERM.
AND n255_02  ; IMP 1Seg.
OUT n50_01  ; TEST.PILOTOS
; rung 9: AVISO LOW BATTERY / ------------------------------------------------------------
LD n253_08  ; LOW BATTERY
ANDNOT nTIM11_STATUS  ; T.AVIS.LOW BATT.
TIM 0010 #100  ; FRCUENC.AVIS.L.B
; rung 10
LD nTIM10_STATUS  ; FRCUENC.AVIS.L.B
TIM 0011 #50  ; T.AVIS.LOW BATT.
; rung 11
LD nTIM10_STATUS  ; FRCUENC.AVIS.L.B
TIM 0012 #2  ; T.CLAXON LOW.BAT
; rung 12
LD nTIM10_STATUS  ; FRCUENC.AVIS.L.B
ANDNOT nTIM11_STATUS  ; T.AVIS.LOW BATT.
OUT n51_00  ; AUX.PILOTO L.B.
; rung 13
LD n51_00  ; AUX.PILOTO L.B.
AND n255_02  ; IMP 1Seg.
OUT n51_01  ; PULSOS LOW BATT.
; rung 14
LD nTIM10_STATUS  ; FRCUENC.AVIS.L.B
ANDNOT nTIM12_STATUS  ; T.CLAXON LOW.BAT
OUT n51_02  ; AUX.CLAXON LOW.B

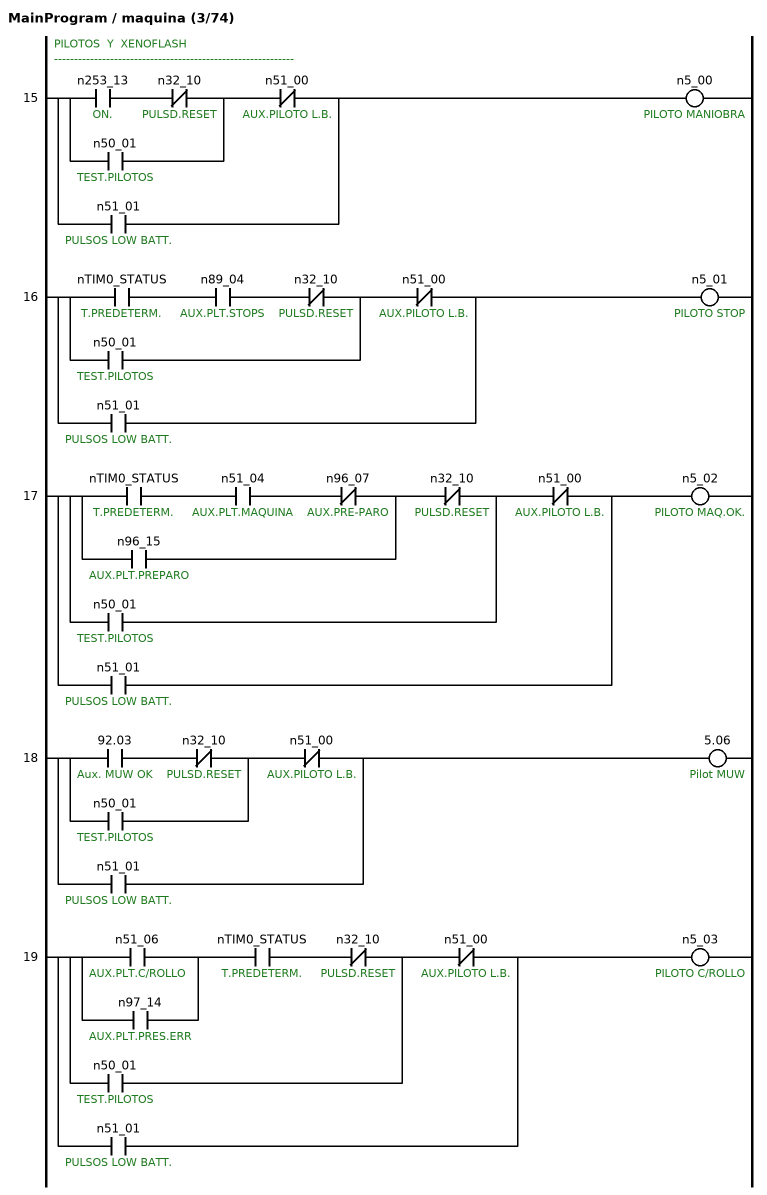
; rung 15: PILOTOS  Y  XENOFLASH / ------------------------------------------------------------
LD n253_13  ; ON.
ANDNOT n32_10  ; PULSD.RESET
OR n50_01  ; TEST.PILOTOS
ANDNOT n51_00  ; AUX.PILOTO L.B.
OR n51_01  ; PULSOS LOW BATT.
OUT n5_00  ; PILOTO MANIOBRA
; rung 16
LD nTIM0_STATUS  ; T.PREDETERM.
AND n89_04  ; AUX.PLT.STOPS
ANDNOT n32_10  ; PULSD.RESET
OR n50_01  ; TEST.PILOTOS
ANDNOT n51_00  ; AUX.PILOTO L.B.
OR n51_01  ; PULSOS LOW BATT.
OUT n5_01  ; PILOTO STOP
; rung 17
LD nTIM0_STATUS  ; T.PREDETERM.
AND n51_04  ; AUX.PLT.MAQUINA
ANDNOT n96_07  ; AUX.PRE-PARO
OR n96_15  ; AUX.PLT.PREPARO
ANDNOT n32_10  ; PULSD.RESET
OR n50_01  ; TEST.PILOTOS
ANDNOT n51_00  ; AUX.PILOTO L.B.
OR n51_01  ; PULSOS LOW BATT.
OUT n5_02  ; PILOTO MAQ.OK.
; rung 18
LD 92.03  ; Aux. MUW OK
ANDNOT n32_10  ; PULSD.RESET
OR n50_01  ; TEST.PILOTOS
ANDNOT n51_00  ; AUX.PILOTO L.B.
OR n51_01  ; PULSOS LOW BATT.
OUT 5.06  ; Pilot MUW
; rung 19
LD n51_06  ; AUX.PLT.C/ROLLO
OR n97_14  ; AUX.PLT.PRES.ERR
AND nTIM0_STATUS  ; T.PREDETERM.
ANDNOT n32_10  ; PULSD.RESET
OR n50_01  ; TEST.PILOTOS
ANDNOT n51_00  ; AUX.PILOTO L.B.
OR n51_01  ; PULSOS LOW BATT.
OUT n5_03  ; PILOTO C/ROLLO

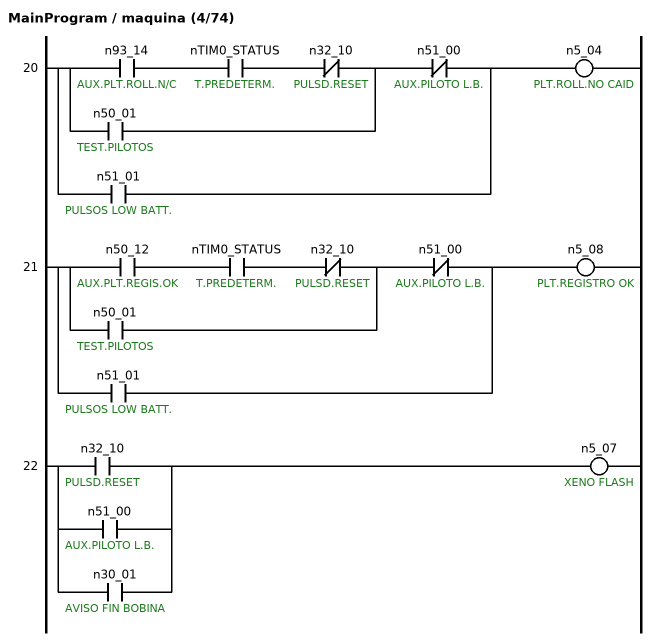
; rung 20
LD n93_14  ; AUX.PLT.ROLL.N/C
AND nTIM0_STATUS  ; T.PREDETERM.
ANDNOT n32_10  ; PULSD.RESET
OR n50_01  ; TEST.PILOTOS
ANDNOT n51_00  ; AUX.PILOTO L.B.
OR n51_01  ; PULSOS LOW BATT.
OUT n5_04  ; PLT.ROLL.NO CAID
; rung 21
LD n50_12  ; AUX.PLT.REGIS.OK
AND nTIM0_STATUS  ; T.PREDETERM.
ANDNOT n32_10  ; PULSD.RESET
OR n50_01  ; TEST.PILOTOS
ANDNOT n51_00  ; AUX.PILOTO L.B.
OR n51_01  ; PULSOS LOW BATT.
OUT n5_08  ; PLT.REGISTRO OK
; rung 22
LD n32_10  ; PULSD.RESET
OR n51_00  ; AUX.PILOTO L.B.
OR n30_01  ; AVISO FIN BOBINA
OUT n5_07  ; XENO FLASH

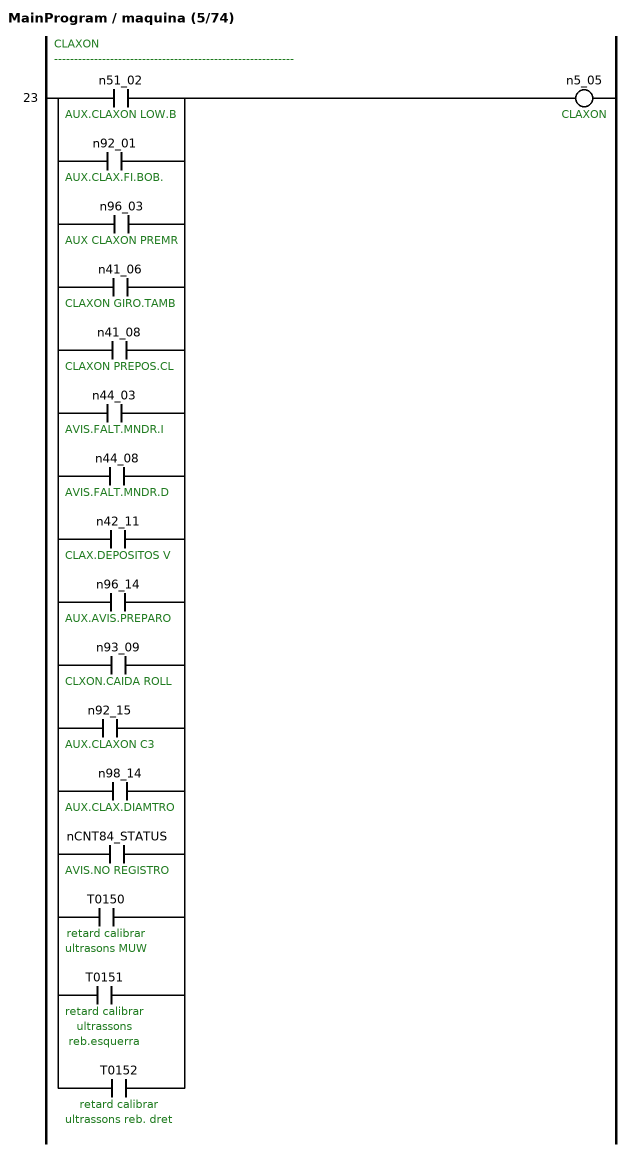
; rung 23: CLAXON / ------------------------------------------------------------
LD n51_02  ; AUX.CLAXON LOW.B
OR n92_01  ; AUX.CLAX.FI.BOB.
OR n96_03  ; AUX CLAXON PREMR
OR n41_06  ; CLAXON GIRO.TAMB
OR n41_08  ; CLAXON PREPOS.CL
OR n44_03  ; AVIS.FALT.MNDR.I
OR n44_08  ; AVIS.FALT.MNDR.D
OR n42_11  ; CLAX.DEPOSITOS V
OR n96_14  ; AUX.AVIS.PREPARO
OR n93_09  ; CLXON.CAIDA ROLL
OR n92_15  ; AUX.CLAXON C3
OR n98_14  ; AUX.CLAX.DIAMTRO
OR nCNT84_STATUS  ; AVIS.NO REGISTRO
OR T0150  ; retard calibrar ultrasons MUW
OR T0151  ; retard calibrar ultrassons reb.esquerra
OR T0152  ; retard calibrar ultrassons reb. dret
OUT n5_05  ; CLAXON

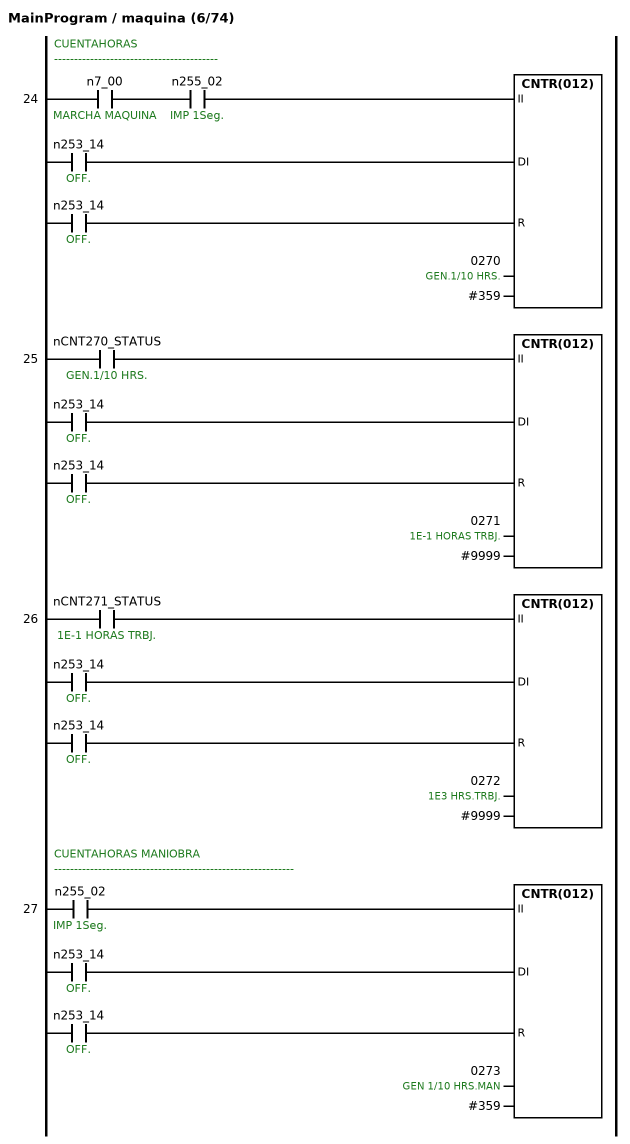
; rung 24: CUENTAHORAS / -----------------------------------------
LD n7_00  ; MARCHA MAQUINA
AND n255_02  ; IMP 1Seg.
LD n253_14  ; OFF.
LD n253_14  ; OFF.
CNTR(012) 0270 #359  ; GEN.1/10 HRS.
; rung 25
LD nCNT270_STATUS  ; GEN.1/10 HRS.
LD n253_14  ; OFF.
LD n253_14  ; OFF.
CNTR(012) 0271 #9999  ; 1E-1 HORAS TRBJ.
; rung 26
LD nCNT271_STATUS  ; 1E-1 HORAS TRBJ.
LD n253_14  ; OFF.
LD n253_14  ; OFF.
CNTR(012) 0272 #9999  ; 1E3 HRS.TRBJ.
; rung 27: CUENTAHORAS MANIOBRA / ------------------------------------------------------------
LD n255_02  ; IMP 1Seg.
LD n253_14  ; OFF.
LD n253_14  ; OFF.
CNTR(012) 0273 #359  ; GEN 1/10 HRS.MAN

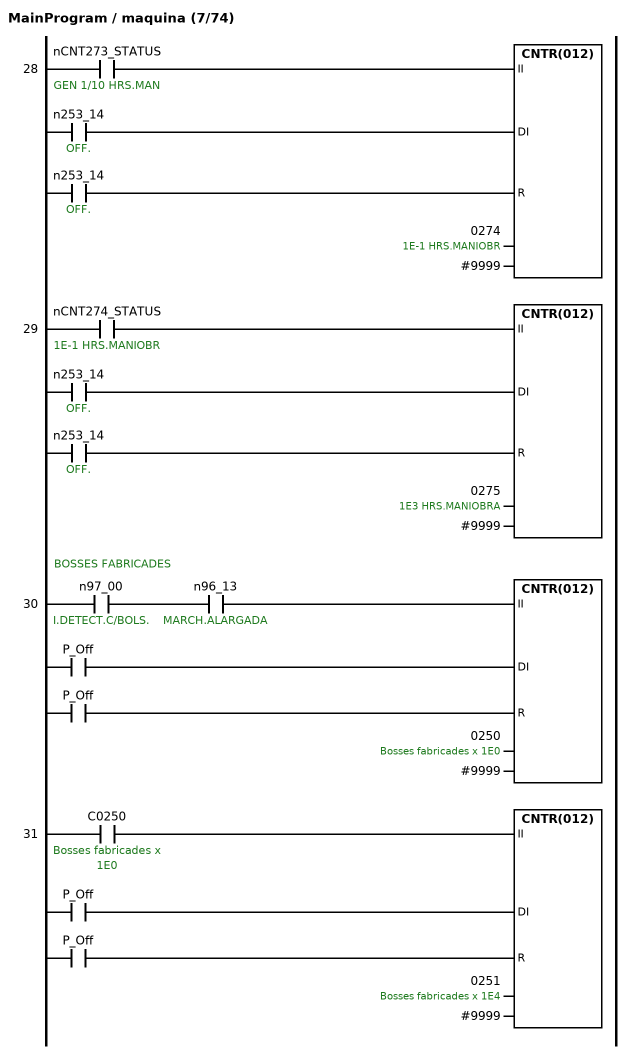
; rung 28
LD nCNT273_STATUS  ; GEN 1/10 HRS.MAN
LD n253_14  ; OFF.
LD n253_14  ; OFF.
CNTR(012) 0274 #9999  ; 1E-1 HRS.MANIOBR
; rung 29
LD nCNT274_STATUS  ; 1E-1 HRS.MANIOBR
LD n253_14  ; OFF.
LD n253_14  ; OFF.
CNTR(012) 0275 #9999  ; 1E3 HRS.MANIOBRA
; rung 30: BOSSES FABRICADES
LD n97_00  ; I.DETECT.C/BOLS.
AND n96_13  ; MARCH.ALARGADA
LD P_Off
LD P_Off
CNTR(012) 0250 #9999  ; Bosses fabricades x 1E0
; rung 31
LD C0250  ; Bosses fabricades x 1E0
LD P_Off
LD P_Off
CNTR(012) 0251 #9999  ; Bosses fabricades x 1E4

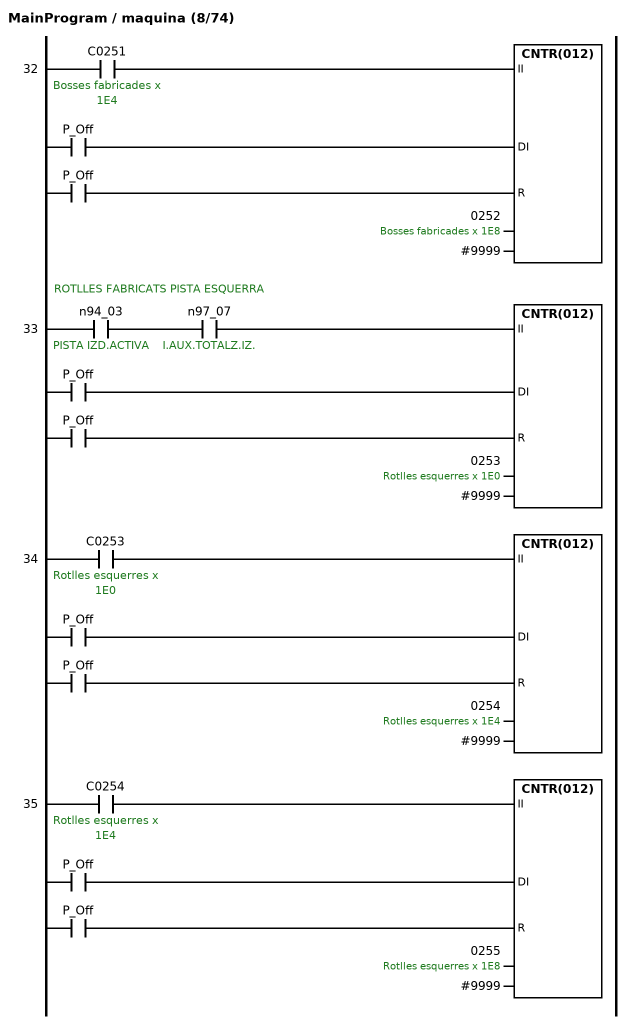
; rung 32
LD C0251  ; Bosses fabricades x 1E4
LD P_Off
LD P_Off
CNTR(012) 0252 #9999  ; Bosses fabricades x 1E8
; rung 33: ROTLLES FABRICATS PISTA ESQUERRA
LD n94_03  ; PISTA IZD.ACTIVA
AND n97_07  ; I.AUX.TOTALZ.IZ.
LD P_Off
LD P_Off
CNTR(012) 0253 #9999  ; Rotlles esquerres x 1E0
; rung 34
LD C0253  ; Rotlles esquerres x 1E0
LD P_Off
LD P_Off
CNTR(012) 0254 #9999  ; Rotlles esquerres x 1E4
; rung 35
LD C0254  ; Rotlles esquerres x 1E4
LD P_Off
LD P_Off
CNTR(012) 0255 #9999  ; Rotlles esquerres x 1E8

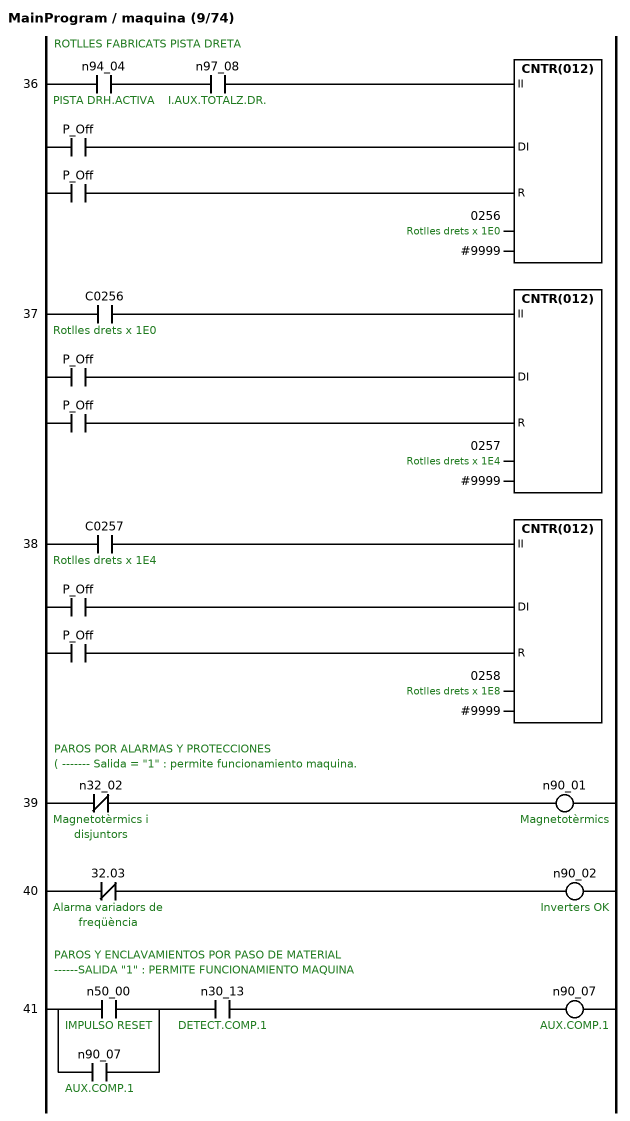
; rung 36: ROTLLES FABRICATS PISTA DRETA
LD n94_04  ; PISTA DRH.ACTIVA
AND n97_08  ; I.AUX.TOTALZ.DR.
LD P_Off
LD P_Off
CNTR(012) 0256 #9999  ; Rotlles drets x 1E0
; rung 37
LD C0256  ; Rotlles drets x 1E0
LD P_Off
LD P_Off
CNTR(012) 0257 #9999  ; Rotlles drets x 1E4
; rung 38
LD C0257  ; Rotlles drets x 1E4
LD P_Off
LD P_Off
CNTR(012) 0258 #9999  ; Rotlles drets x 1E8
; rung 39: PAROS POR ALARMAS Y PROTECCIONES / ( ------- Salida = "1" : permite funcionamiento maquina.
LDNOT n32_02  ; Magnetotèrmics i disjuntors
OUT n90_01  ; Magnetotèrmics
; rung 40
LDNOT 32.03  ; Alarma variadors de freqüència
OUT n90_02  ; Inverters OK
; rung 41: PAROS Y ENCLAVAMIENTOS POR PASO DE MATERIAL / ------SALIDA "1" : PERMITE FUNCIONAMIENTO MAQUINA
LD n50_00  ; IMPULSO RESET
OR n90_07  ; AUX.COMP.1
AND n30_13  ; DETECT.COMP.1
OUT n90_07  ; AUX.COMP.1

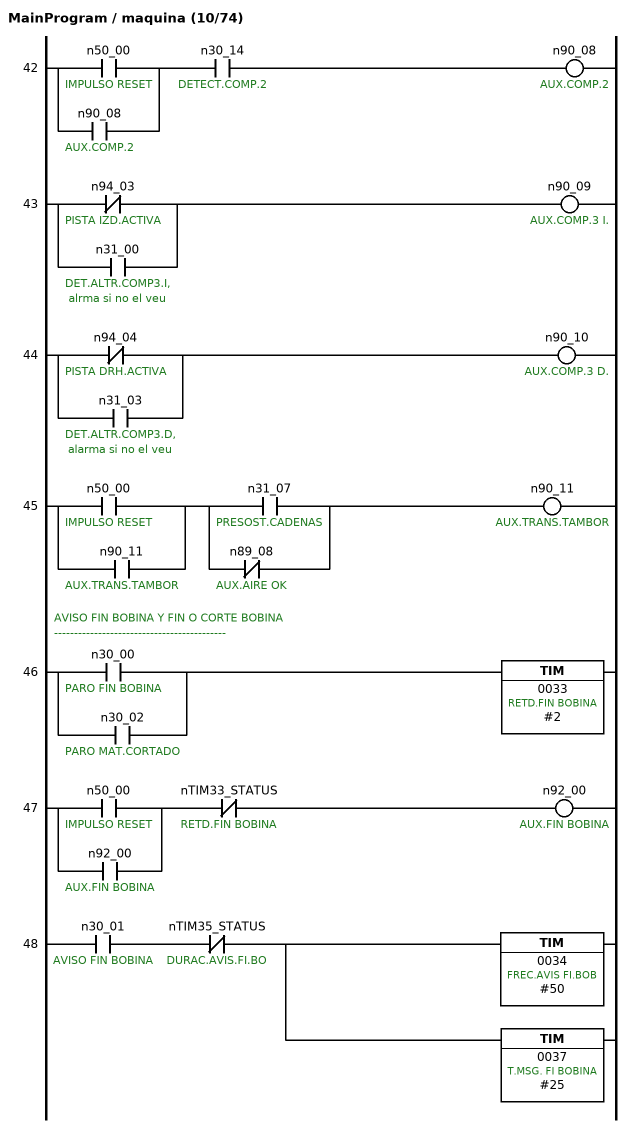
; rung 42
LD n50_00  ; IMPULSO RESET
OR n90_08  ; AUX.COMP.2
AND n30_14  ; DETECT.COMP.2
OUT n90_08  ; AUX.COMP.2
; rung 43
LDNOT n94_03  ; PISTA IZD.ACTIVA
OR n31_00  ; DET.ALTR.COMP3.I, alrma si no el veu
OUT n90_09  ; AUX.COMP.3 I.
; rung 44
LDNOT n94_04  ; PISTA DRH.ACTIVA
OR n31_03  ; DET.ALTR.COMP3.D, alarma si no el veu
OUT n90_10  ; AUX.COMP.3 D.
; rung 45
LD n50_00  ; IMPULSO RESET
OR n90_11  ; AUX.TRANS.TAMBOR
LD n31_07  ; PRESOST.CADENAS
ORNOT n89_08  ; AUX.AIRE OK
ANDLD
OUT n90_11  ; AUX.TRANS.TAMBOR
; rung 46: AVISO FIN BOBINA Y FIN O CORTE BOBINA / -------------------------------------------
LD n30_00  ; PARO FIN BOBINA
OR n30_02  ; PARO MAT.CORTADO
TIM 0033 #2  ; RETD.FIN BOBINA
; rung 47
LD n50_00  ; IMPULSO RESET
OR n92_00  ; AUX.FIN BOBINA
ANDNOT nTIM33_STATUS  ; RETD.FIN BOBINA
OUT n92_00  ; AUX.FIN BOBINA
; rung 48
LD n30_01  ; AVISO FIN BOBINA
ANDNOT nTIM35_STATUS  ; DURAC.AVIS.FI.BO
TIM 0034 #50  ; FREC.AVIS FI.BOB
TIM 0037 #25  ; T.MSG. FI BOBINA

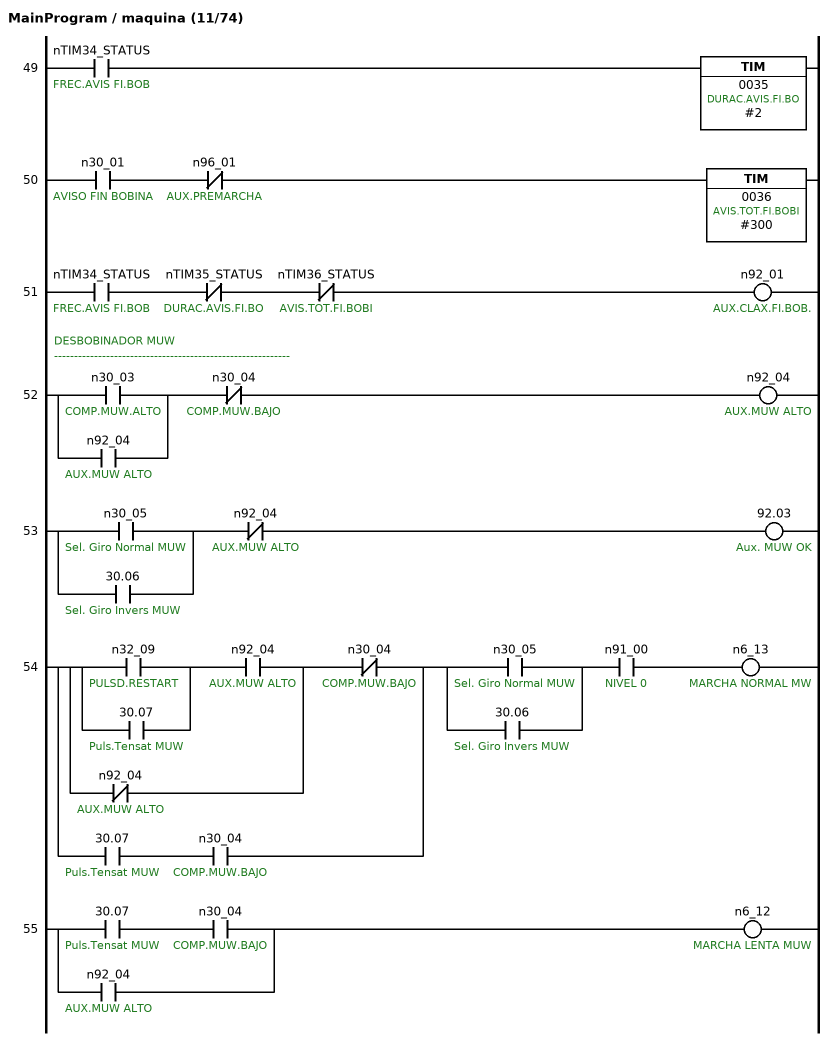
; rung 49
LD nTIM34_STATUS  ; FREC.AVIS FI.BOB
TIM 0035 #2  ; DURAC.AVIS.FI.BO
; rung 50
LD n30_01  ; AVISO FIN BOBINA
ANDNOT n96_01  ; AUX.PREMARCHA
TIM 0036 #300  ; AVIS.TOT.FI.BOBI
; rung 51
LD nTIM34_STATUS  ; FREC.AVIS FI.BOB
ANDNOT nTIM35_STATUS  ; DURAC.AVIS.FI.BO
ANDNOT nTIM36_STATUS  ; AVIS.TOT.FI.BOBI
OUT n92_01  ; AUX.CLAX.FI.BOB.
; rung 52: DESBOBINADOR MUW / -----------------------------------------------------------
LD n30_03  ; COMP.MUW.ALTO
OR n92_04  ; AUX.MUW ALTO
ANDNOT n30_04  ; COMP.MUW.BAJO
OUT n92_04  ; AUX.MUW ALTO
; rung 53
LD n30_05  ; Sel. Giro Normal MUW
OR 30.06  ; Sel. Giro Invers MUW
ANDNOT n92_04  ; AUX.MUW ALTO
OUT 92.03  ; Aux. MUW OK
; rung 54
LD n32_09  ; PULSD.RESTART
OR 30.07  ; Puls.Tensat MUW
AND n92_04  ; AUX.MUW ALTO
ORNOT n92_04  ; AUX.MUW ALTO
ANDNOT n30_04  ; COMP.MUW.BAJO
LD 30.07  ; Puls.Tensat MUW
AND n30_04  ; COMP.MUW.BAJO
ORLD
LD n30_05  ; Sel. Giro Normal MUW
OR 30.06  ; Sel. Giro Invers MUW
ANDLD
AND n91_00  ; NIVEL 0
OUT n6_13  ; MARCHA NORMAL MW
; rung 55
LD 30.07  ; Puls.Tensat MUW
AND n30_04  ; COMP.MUW.BAJO
OR n92_04  ; AUX.MUW ALTO
OUT n6_12  ; MARCHA LENTA MUW

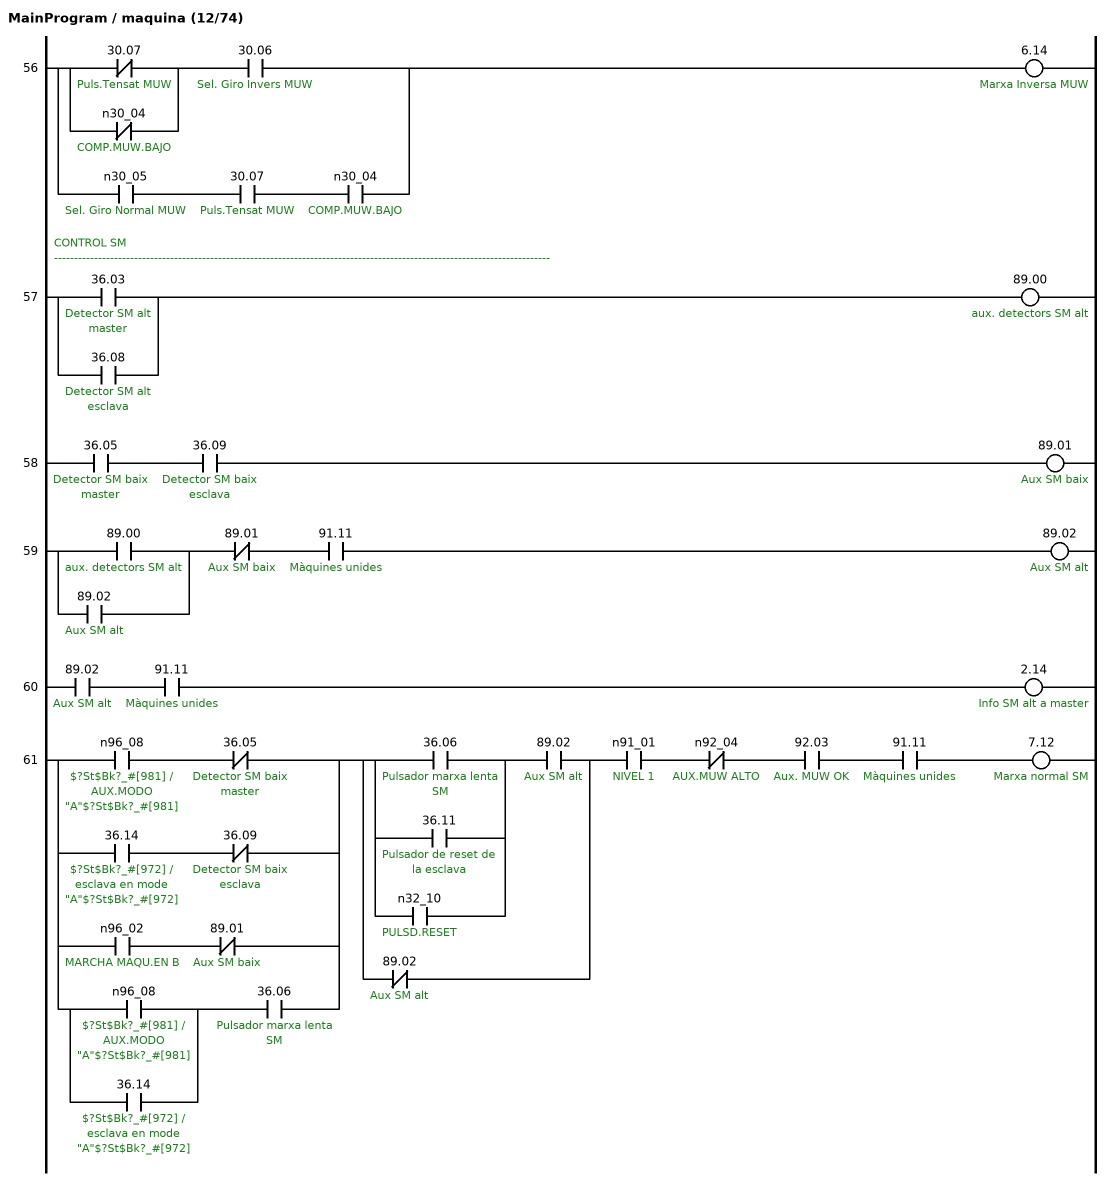
; rung 56
LDNOT 30.07  ; Puls.Tensat MUW
ORNOT n30_04  ; COMP.MUW.BAJO
AND 30.06  ; Sel. Giro Invers MUW
LD n30_05  ; Sel. Giro Normal MUW
AND 30.07  ; Puls.Tensat MUW
AND n30_04  ; COMP.MUW.BAJO
ORLD
OUT 6.14  ; Marxa Inversa MUW
; rung 57: CONTROL SM / ----------------------------------------------------------------------------------------------------------------------------
LD 36.03  ; Detector SM alt master
OR 36.08  ; Detector SM alt esclava
OUT 89.00  ; aux. detectors SM alt
; rung 58
LD 36.05  ; Detector SM baix master
AND 36.09  ; Detector SM baix esclava
OUT 89.01  ; Aux SM baix
; rung 59
LD 89.00  ; aux. detectors SM alt
OR 89.02  ; Aux SM alt
ANDNOT 89.01  ; Aux SM baix
AND 91.11  ; Màquines unides
OUT 89.02  ; Aux SM alt
; rung 60
LD 89.02  ; Aux SM alt
AND 91.11  ; Màquines unides
OUT 2.14  ; Info SM alt a master
; rung 61
LD n96_08  ; $?St$Bk?_#[981] / AUX.MODO "A"$?St$Bk?_#[981]
ANDNOT 36.05  ; Detector SM baix master
LD 36.14  ; $?St$Bk?_#[972] / esclava en mode "A"$?St$Bk?_#[972]
ANDNOT 36.09  ; Detector SM baix esclava
ORLD
LD n96_02  ; MARCHA MAQU.EN B
ANDNOT 89.01  ; Aux SM baix
ORLD
LD n96_08  ; $?St$Bk?_#[981] / AUX.MODO "A"$?St$Bk?_#[981]
OR 36.14  ; $?St$Bk?_#[972] / esclava en mode "A"$?St$Bk?_#[972]
AND 36.06  ; Pulsador marxa lenta SM
ORLD
LD 36.06  ; Pulsador marxa lenta SM
OR 36.11  ; Pulsador de reset de la esclava
OR n32_10  ; PULSD.RESET
AND 89.02  ; Aux SM alt
ORNOT 89.02  ; Aux SM alt
ANDLD
AND n91_01  ; NIVEL 1
ANDNOT n92_04  ; AUX.MUW ALTO
AND 92.03  ; Aux. MUW OK
AND 91.11  ; Màquines unides
OUT 7.12  ; Marxa normal SM

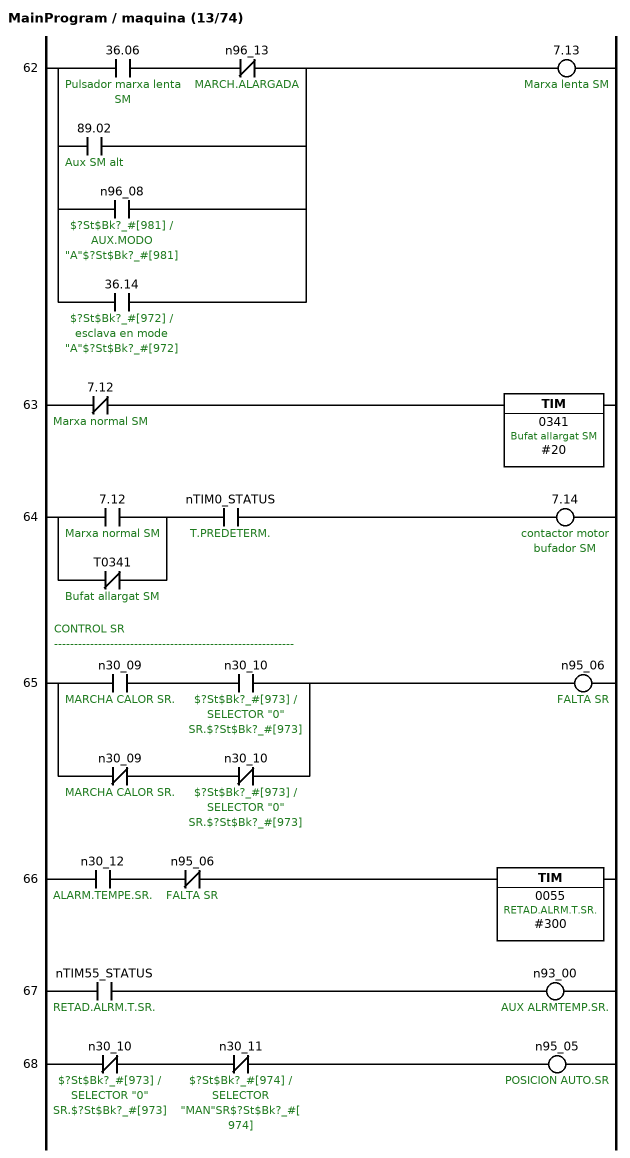
; rung 62
LD 36.06  ; Pulsador marxa lenta SM
ANDNOT n96_13  ; MARCH.ALARGADA
OR 89.02  ; Aux SM alt
OR n96_08  ; $?St$Bk?_#[981] / AUX.MODO "A"$?St$Bk?_#[981]
OR 36.14  ; $?St$Bk?_#[972] / esclava en mode "A"$?St$Bk?_#[972]
OUT 7.13  ; Marxa lenta SM
; rung 63
LDNOT 7.12  ; Marxa normal SM
TIM 0341 #20  ; Bufat allargat SM
; rung 64
LD 7.12  ; Marxa normal SM
ORNOT T0341  ; Bufat allargat SM
AND nTIM0_STATUS  ; T.PREDETERM.
OUT 7.14  ; contactor motor bufador SM
; rung 65: CONTROL SR / ------------------------------------------------------------
LD n30_09  ; MARCHA CALOR SR.
AND n30_10  ; $?St$Bk?_#[973] / SELECTOR "0" SR.$?St$Bk?_#[973]
LDNOT n30_09  ; MARCHA CALOR SR.
ANDNOT n30_10  ; $?St$Bk?_#[973] / SELECTOR "0" SR.$?St$Bk?_#[973]
ORLD
OUT n95_06  ; FALTA SR
; rung 66
LD n30_12  ; ALARM.TEMPE.SR.
ANDNOT n95_06  ; FALTA SR
TIM 0055 #300  ; RETAD.ALRM.T.SR.
; rung 67
LD nTIM55_STATUS  ; RETAD.ALRM.T.SR.
OUT n93_00  ; AUX ALRMTEMP.SR.
; rung 68
LDNOT n30_10  ; $?St$Bk?_#[973] / SELECTOR "0" SR.$?St$Bk?_#[973]
ANDNOT n30_11  ; $?St$Bk?_#[974] / SELECTOR "MAN"SR$?St$Bk?_#[974]
OUT n95_05  ; POSICION AUTO.SR

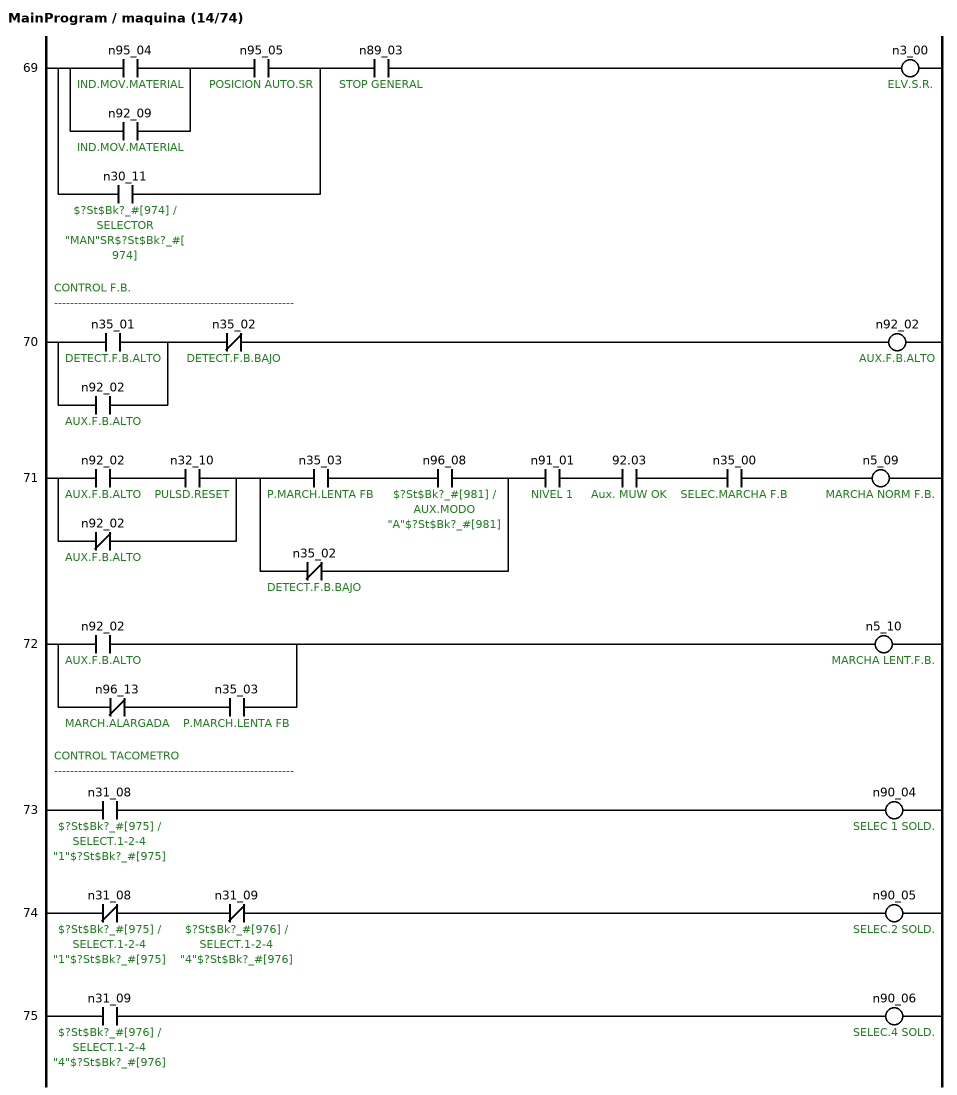
; rung 69
LD n95_04  ; IND.MOV.MATERIAL
OR n92_09  ; IND.MOV.MATERIAL
AND n95_05  ; POSICION AUTO.SR
OR n30_11  ; $?St$Bk?_#[974] / SELECTOR "MAN"SR$?St$Bk?_#[974]
AND n89_03  ; STOP GENERAL
OUT n3_00  ; ELV.S.R.
; rung 70: CONTROL F.B. / ------------------------------------------------------------
LD n35_01  ; DETECT.F.B.ALTO
OR n92_02  ; AUX.F.B.ALTO
ANDNOT n35_02  ; DETECT.F.B.BAJO
OUT n92_02  ; AUX.F.B.ALTO
; rung 71
LD n92_02  ; AUX.F.B.ALTO
AND n32_10  ; PULSD.RESET
ORNOT n92_02  ; AUX.F.B.ALTO
LD n35_03  ; P.MARCH.LENTA FB
AND n96_08  ; $?St$Bk?_#[981] / AUX.MODO "A"$?St$Bk?_#[981]
ORNOT n35_02  ; DETECT.F.B.BAJO
ANDLD
AND n91_01  ; NIVEL 1
AND 92.03  ; Aux. MUW OK
AND n35_00  ; SELEC.MARCHA F.B
OUT n5_09  ; MARCHA NORM F.B.
; rung 72
LD n92_02  ; AUX.F.B.ALTO
LDNOT n96_13  ; MARCH.ALARGADA
AND n35_03  ; P.MARCH.LENTA FB
ORLD
OUT n5_10  ; MARCHA LENT.F.B.
; rung 73: CONTROL TACOMETRO / ------------------------------------------------------------
LD n31_08  ; $?St$Bk?_#[975] / SELECT.1-2-4 "1"$?St$Bk?_#[975]
OUT n90_04  ; SELEC 1 SOLD.
; rung 74
LDNOT n31_08  ; $?St$Bk?_#[975] / SELECT.1-2-4 "1"$?St$Bk?_#[975]
ANDNOT n31_09  ; $?St$Bk?_#[976] / SELECT.1-2-4 "4"$?St$Bk?_#[976]
OUT n90_05  ; SELEC.2 SOLD.
; rung 75
LD n31_09  ; $?St$Bk?_#[976] / SELECT.1-2-4 "4"$?St$Bk?_#[976]
OUT n90_06  ; SELEC.4 SOLD.

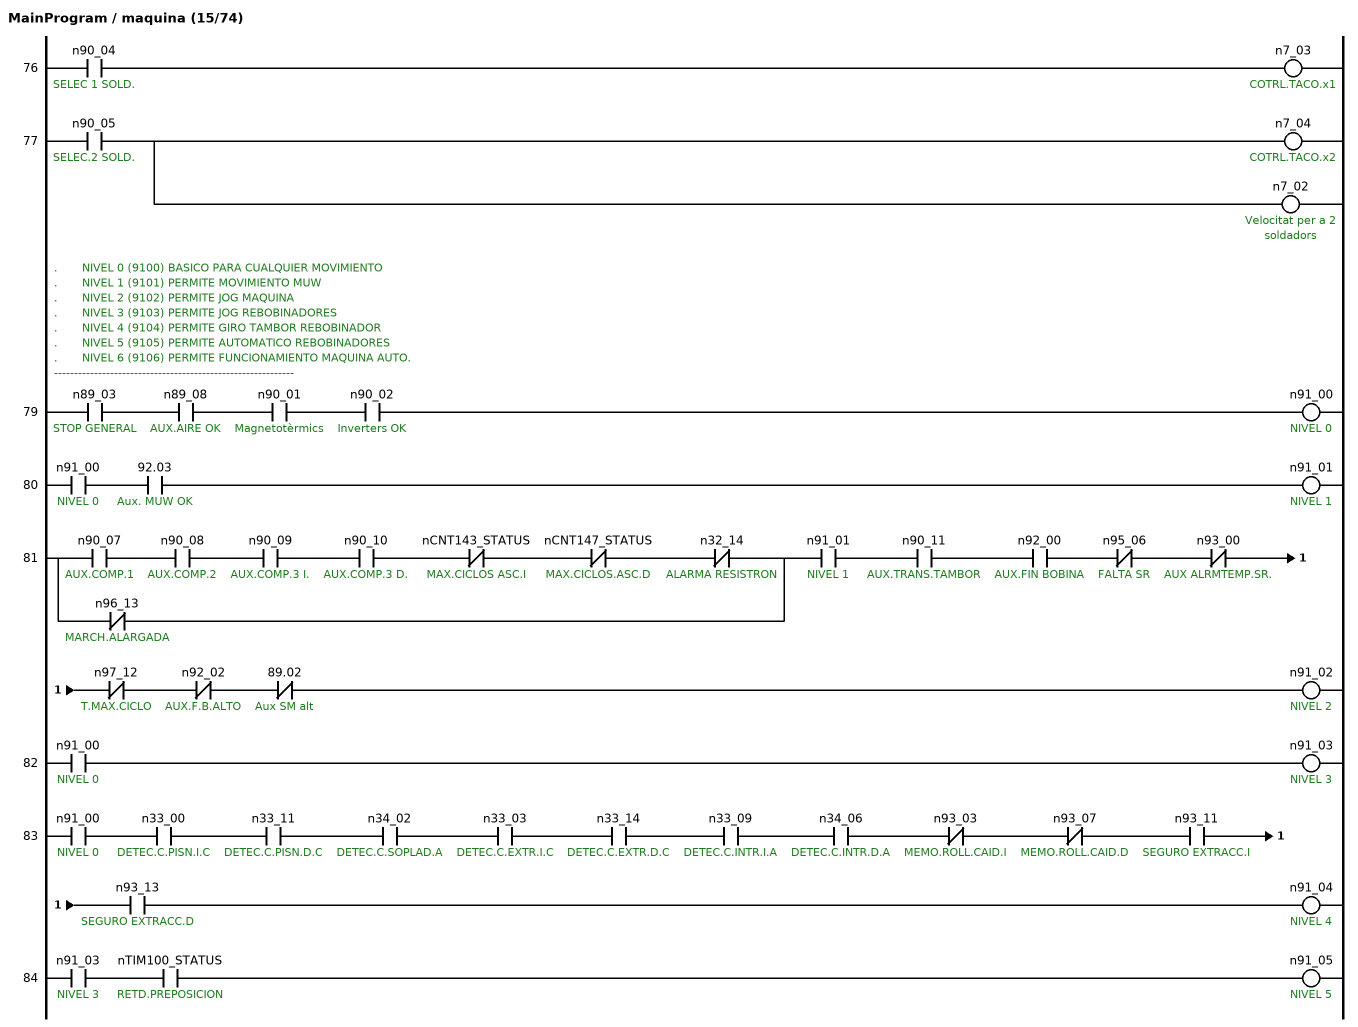
; rung 76
LD n90_04  ; SELEC 1 SOLD.
OUT n7_03  ; COTRL.TACO.x1
; rung 77
LD n90_05  ; SELEC.2 SOLD.
OUT n7_04  ; COTRL.TACO.x2
OUT n7_02  ; Velocitat per a 2 soldadors
; rung 78: DETERMINACION DE NIVELES DE PERMISION DE MOVIMIENTOS / ************************************************************
; rung 79: .       NIVEL 0 (9100) BASICO PARA CUALQUIER MOVIMIENTO / .       NIVEL 1 (9101) PERMITE MOVIMIENTO MUW / .       NIVEL 2 (9102) PERMITE JOG MAQUINA / .       NIVEL 3 (9103) PERMITE JOG REBOBINADORES / .       NIVEL 4 (9104) PERMITE GIRO TAMBOR REBOBINADOR / .       NIVEL 5 (9105) PERMITE AUTOMATICO REBOBINADORES / .       NIVEL 6 (9106) PERMITE FUNCIONAMIENTO MAQUINA AUTO. / ------------------------------------------------------------
LD n89_03  ; STOP GENERAL
AND n89_08  ; AUX.AIRE OK
AND n90_01  ; Magnetotèrmics
AND n90_02  ; Inverters OK
OUT n91_00  ; NIVEL 0
; rung 80
LD n91_00  ; NIVEL 0
AND 92.03  ; Aux. MUW OK
OUT n91_01  ; NIVEL 1
; rung 81
LD n90_07  ; AUX.COMP.1
AND n90_08  ; AUX.COMP.2
AND n90_09  ; AUX.COMP.3 I.
AND n90_10  ; AUX.COMP.3 D.
ANDNOT nCNT143_STATUS  ; MAX.CICLOS ASC.I
ANDNOT nCNT147_STATUS  ; MAX.CICLOS.ASC.D
ANDNOT n32_14  ; ALARMA RESISTRON
ORNOT n96_13  ; MARCH.ALARGADA
AND n91_01  ; NIVEL 1
AND n90_11  ; AUX.TRANS.TAMBOR
AND n92_00  ; AUX.FIN BOBINA
ANDNOT n95_06  ; FALTA SR
ANDNOT n93_00  ; AUX ALRMTEMP.SR.
ANDNOT n97_12  ; T.MAX.CICLO
ANDNOT n92_02  ; AUX.F.B.ALTO
ANDNOT 89.02  ; Aux SM alt
OUT n91_02  ; NIVEL 2
; rung 82
LD n91_00  ; NIVEL 0
OUT n91_03  ; NIVEL 3
; rung 83
LD n91_00  ; NIVEL 0
AND n33_00  ; DETEC.C.PISN.I.C
AND n33_11  ; DETEC.C.PISN.D.C
AND n34_02  ; DETEC.C.SOPLAD.A
AND n33_03  ; DETEC.C.EXTR.I.C
AND n33_14  ; DETEC.C.EXTR.D.C
AND n33_09  ; DETEC.C.INTR.I.A
AND n34_06  ; DETEC.C.INTR.D.A
ANDNOT n93_03  ; MEMO.ROLL.CAID.I
ANDNOT n93_07  ; MEMO.ROLL.CAID.D
AND n93_11  ; SEGURO EXTRACC.I
AND n93_13  ; SEGURO EXTRACC.D
OUT n91_04  ; NIVEL 4
; rung 84
LD n91_03  ; NIVEL 3
AND nTIM100_STATUS  ; RETD.PREPOSICION
OUT n91_05  ; NIVEL 5

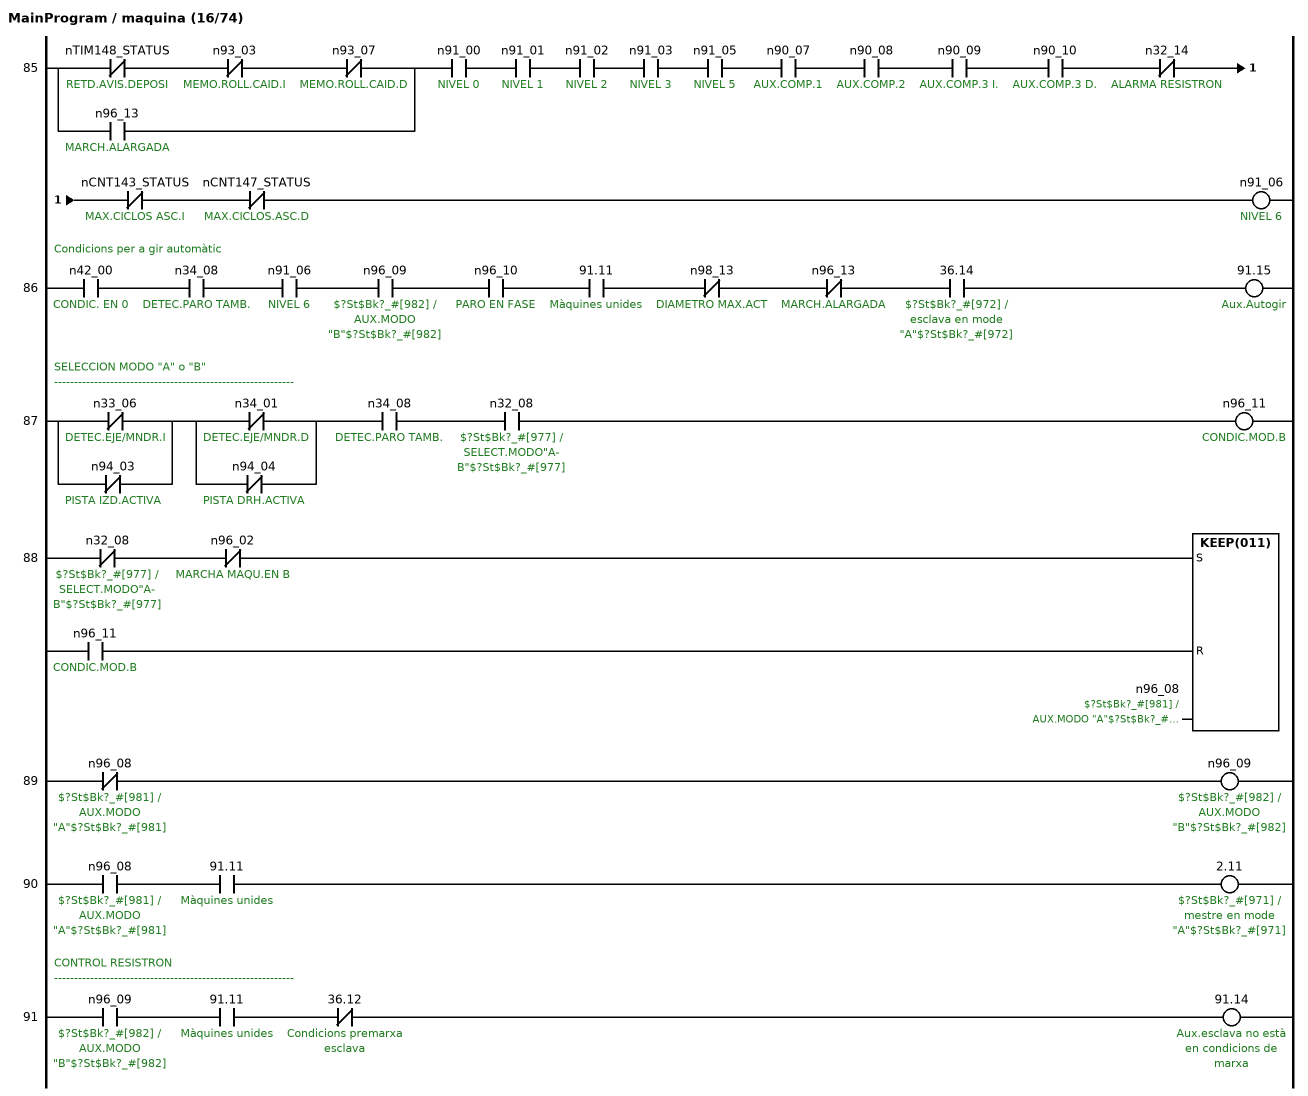
; rung 85
LDNOT nTIM148_STATUS  ; RETD.AVIS.DEPOSI
ANDNOT n93_03  ; MEMO.ROLL.CAID.I
ANDNOT n93_07  ; MEMO.ROLL.CAID.D
OR n96_13  ; MARCH.ALARGADA
AND n91_00  ; NIVEL 0
AND n91_01  ; NIVEL 1
AND n91_02  ; NIVEL 2
AND n91_03  ; NIVEL 3
AND n91_05  ; NIVEL 5
AND n90_07  ; AUX.COMP.1
AND n90_08  ; AUX.COMP.2
AND n90_09  ; AUX.COMP.3 I.
AND n90_10  ; AUX.COMP.3 D.
ANDNOT n32_14  ; ALARMA RESISTRON
ANDNOT nCNT143_STATUS  ; MAX.CICLOS ASC.I
ANDNOT nCNT147_STATUS  ; MAX.CICLOS.ASC.D
OUT n91_06  ; NIVEL 6
; rung 86: Condicions per a gir automàtic
LD n42_00  ; CONDIC. EN 0
AND n34_08  ; DETEC.PARO TAMB.
AND n91_06  ; NIVEL 6
AND n96_09  ; $?St$Bk?_#[982] / AUX.MODO "B"$?St$Bk?_#[982]
AND n96_10  ; PARO EN FASE
AND 91.11  ; Màquines unides
ANDNOT n98_13  ; DIAMETRO MAX.ACT
ANDNOT n96_13  ; MARCH.ALARGADA
AND 36.14  ; $?St$Bk?_#[972] / esclava en mode "A"$?St$Bk?_#[972]
OUT 91.15  ; Aux.Autogir
; rung 87: SELECCION MODO "A" o "B" / ------------------------------------------------------------
LDNOT n33_06  ; DETEC.EJE/MNDR.I
ORNOT n94_03  ; PISTA IZD.ACTIVA
LDNOT n34_01  ; DETEC.EJE/MNDR.D
ORNOT n94_04  ; PISTA DRH.ACTIVA
ANDLD
AND n34_08  ; DETEC.PARO TAMB.
AND n32_08  ; $?St$Bk?_#[977] / SELECT.MODO"A-B"$?St$Bk?_#[977]
OUT n96_11  ; CONDIC.MOD.B
; rung 88
LDNOT n32_08  ; $?St$Bk?_#[977] / SELECT.MODO"A-B"$?St$Bk?_#[977]
ANDNOT n96_02  ; MARCHA MAQU.EN B
LD n96_11  ; CONDIC.MOD.B
KEEP(011) n96_08  ; $?St$Bk?_#[981] / AUX.MODO "A"$?St$Bk?_#[981]
; rung 89
LDNOT n96_08  ; $?St$Bk?_#[981] / AUX.MODO "A"$?St$Bk?_#[981]
OUT n96_09  ; $?St$Bk?_#[982] / AUX.MODO "B"$?St$Bk?_#[982]
; rung 90
LD n96_08  ; $?St$Bk?_#[981] / AUX.MODO "A"$?St$Bk?_#[981]
AND 91.11  ; Màquines unides
OUT 2.11  ; $?St$Bk?_#[971] / mestre en mode "A"$?St$Bk?_#[971]
; rung 91: CONTROL RESISTRON / ------------------------------------------------------------
LD n96_09  ; $?St$Bk?_#[982] / AUX.MODO "B"$?St$Bk?_#[982]
AND 91.11  ; Màquines unides
ANDNOT 36.12  ; Condicions premarxa esclava
OUT 91.14  ; Aux.esclava no està en condicions de marxa

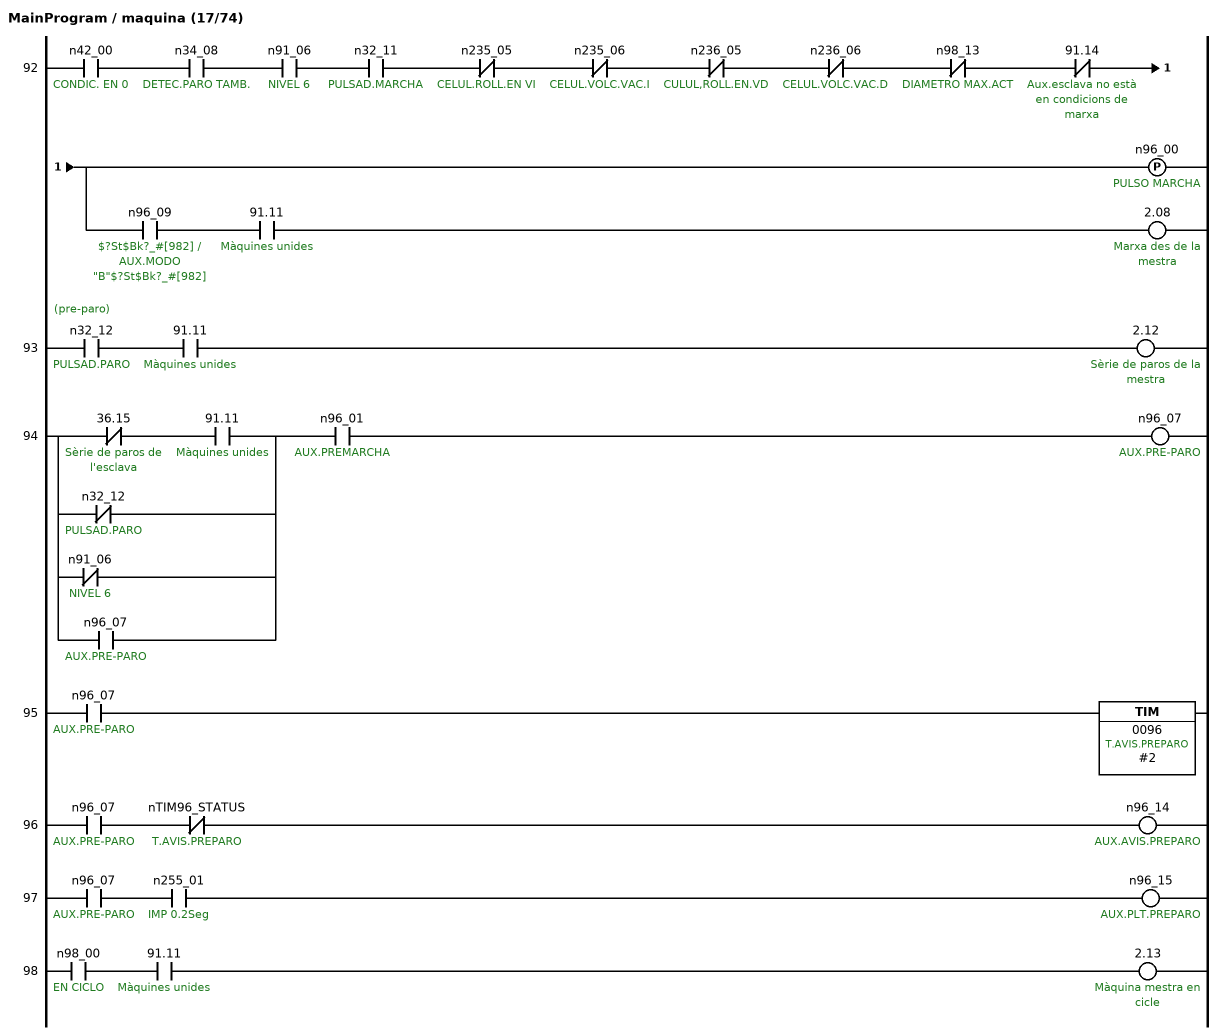
; rung 92
LD n42_00  ; CONDIC. EN 0
AND n34_08  ; DETEC.PARO TAMB.
AND n91_06  ; NIVEL 6
AND n32_11  ; PULSAD.MARCHA
ANDNOT n235_05  ; CELUL.ROLL.EN VI
ANDNOT n235_06  ; CELUL.VOLC.VAC.I
ANDNOT n236_05  ; CULUL,ROLL.EN.VD
ANDNOT n236_06  ; CELUL.VOLC.VAC.D
ANDNOT n98_13  ; DIAMETRO MAX.ACT
ANDNOT 91.14  ; Aux.esclava no està en condicions de marxa
DIFU(013) n96_00  ; PULSO MARCHA
AND n96_09  ; $?St$Bk?_#[982] / AUX.MODO "B"$?St$Bk?_#[982]
AND 91.11  ; Màquines unides
OUT 2.08  ; Marxa des de la mestra
; rung 93: (pre-paro)
LD n32_12  ; PULSAD.PARO
AND 91.11  ; Màquines unides
OUT 2.12  ; Sèrie de paros de la mestra
; rung 94
LDNOT 36.15  ; Sèrie de paros de l'esclava
AND 91.11  ; Màquines unides
ORNOT n32_12  ; PULSAD.PARO
ORNOT n91_06  ; NIVEL 6
OR n96_07  ; AUX.PRE-PARO
AND n96_01  ; AUX.PREMARCHA
OUT n96_07  ; AUX.PRE-PARO
; rung 95
LD n96_07  ; AUX.PRE-PARO
TIM 0096 #2  ; T.AVIS.PREPARO
; rung 96
LD n96_07  ; AUX.PRE-PARO
ANDNOT nTIM96_STATUS  ; T.AVIS.PREPARO
OUT n96_14  ; AUX.AVIS.PREPARO
; rung 97
LD n96_07  ; AUX.PRE-PARO
AND n255_01  ; IMP 0.2Seg
OUT n96_15  ; AUX.PLT.PREPARO
; rung 98
LD n98_00  ; EN CICLO
AND 91.11  ; Màquines unides
OUT 2.13  ; Màquina mestra en cicle

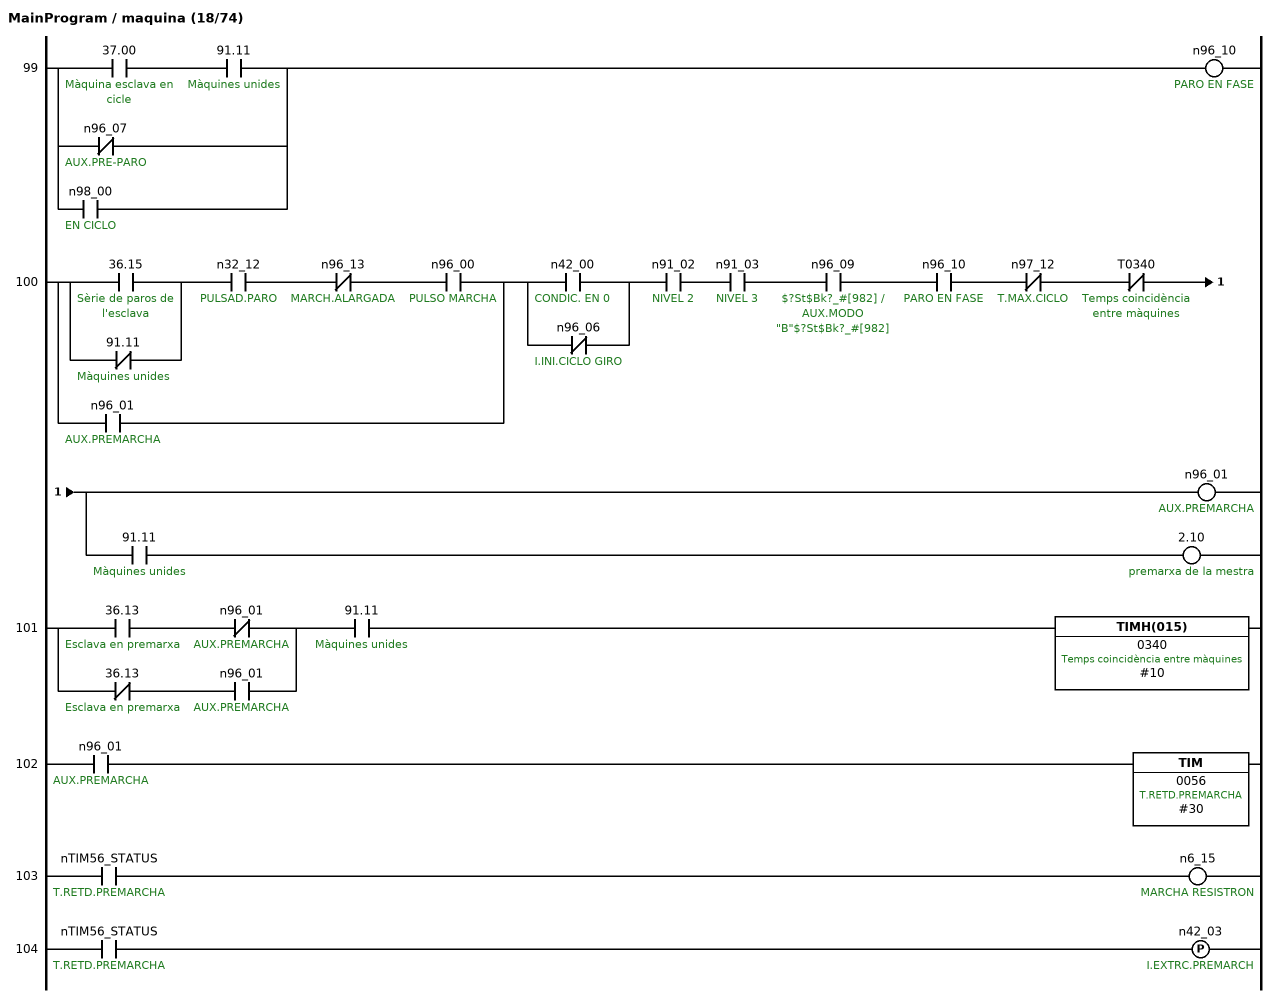
; rung 99
LD 37.00  ; Màquina esclava en cicle
AND 91.11  ; Màquines unides
ORNOT n96_07  ; AUX.PRE-PARO
OR n98_00  ; EN CICLO
OUT n96_10  ; PARO EN FASE
; rung 100
LD 36.15  ; Sèrie de paros de l'esclava
ORNOT 91.11  ; Màquines unides
AND n32_12  ; PULSAD.PARO
ANDNOT n96_13  ; MARCH.ALARGADA
AND n96_00  ; PULSO MARCHA
OR n96_01  ; AUX.PREMARCHA
LD n42_00  ; CONDIC. EN 0
ORNOT n96_06  ; I.INI.CICLO GIRO
ANDLD
AND n91_02  ; NIVEL 2
AND n91_03  ; NIVEL 3
AND n96_09  ; $?St$Bk?_#[982] / AUX.MODO "B"$?St$Bk?_#[982]
AND n96_10  ; PARO EN FASE
ANDNOT n97_12  ; T.MAX.CICLO
ANDNOT T0340  ; Temps coincidència entre màquines
OUT n96_01  ; AUX.PREMARCHA
AND 91.11  ; Màquines unides
OUT 2.10  ; premarxa de la mestra
; rung 101
LD 36.13  ; Esclava en premarxa
ANDNOT n96_01  ; AUX.PREMARCHA
LDNOT 36.13  ; Esclava en premarxa
AND n96_01  ; AUX.PREMARCHA
ORLD
AND 91.11  ; Màquines unides
TIMH(015) 0340 #10  ; Temps coincidència entre màquines
; rung 102
LD n96_01  ; AUX.PREMARCHA
TIM 0056 #30  ; T.RETD.PREMARCHA
; rung 103
LD nTIM56_STATUS  ; T.RETD.PREMARCHA
OUT n6_15  ; MARCHA RESISTRON
; rung 104
LD nTIM56_STATUS  ; T.RETD.PREMARCHA
DIFU(013) n42_03  ; I.EXTRC.PREMARCH

